METHOD PRIVATE M_MotionDynamicMove
VAR_INPUT
END_VAR
VAR_INST
	{attribute 'tc_no_symbol'}                	                			
	_fb_MovePosDynamic			: ARRAY [1..4] OF FB_ServoMotionDynamics;
	{attribute 'tc_no_symbol'}                	                			
	_enableDynamicMove			: BOOL;
	{attribute 'tc_no_symbol'}                	                			
	_Pos2MoveStart				: ST_MovePosition_SP;
	{attribute 'tc_no_symbol'}                	                			
	_CMD_MoveDynamicAbsStart	: ARRAY[1..4] OF MC_MOVEABSOLUTE;
	{attribute 'tc_no_symbol'}                	                			
	_CMD_MoveDynamicAbsEnd		: ARRAY[1..4] OF MC_MOVEABSOLUTE;
END_VAR
VAR_INST // added by the converter: edge detectors and wires of the graphical bodies
    _rt1, _rt2, _rt3, _rt4, _rt5, _rt6, _rt7, _rt8, _rt9, _rt10 : R_TRIG;
    _w1, _w2 : BOOL;
END_VAR
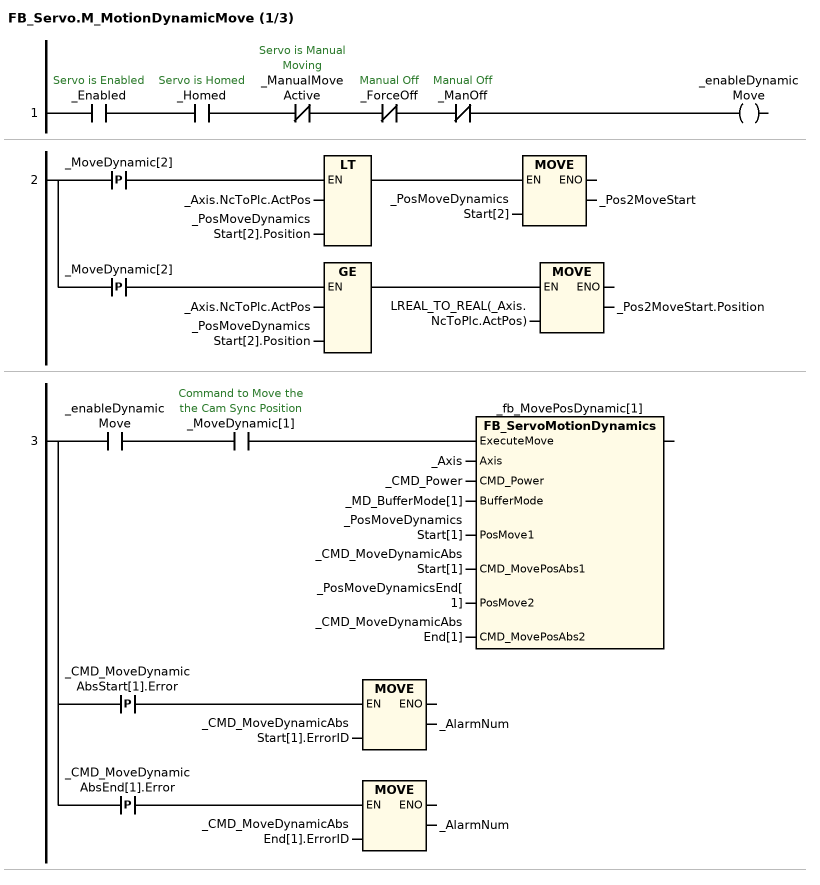
// NETWORK 1
//   _Enabled: Servo is Enabled
//   _Homed: Servo is Homed
//   _ManualMoveActive: Servo is Manual Moving
//   _ForceOff: Manual Off
//   _ManOff: Manual Off
_enableDynamicMove := _Enabled AND _Homed AND NOT _ManualMoveActive AND NOT _ForceOff AND NOT _ManOff;

// NETWORK 2
_rt1(CLK := _MoveDynamic[2]);
_w1 := _rt1.Q AND _Axis.NcToPlc.ActPos < _PosMoveDynamicsStart[2].Position;
IF _w1 THEN _Pos2MoveStart := _PosMoveDynamicsStart[2]; END_IF
_rt2(CLK := _MoveDynamic[2]);
_w2 := _rt2.Q AND _Axis.NcToPlc.ActPos >= _PosMoveDynamicsStart[2].Position;
IF _w2 THEN _Pos2MoveStart.Position := LREAL_TO_REAL(_Axis.NcToPlc.ActPos); END_IF

// NETWORK 3
//   _MoveDynamic[1]: Command to Move the the Cam Sync Position
_fb_MovePosDynamic[1](
    ExecuteMove := _enableDynamicMove AND _MoveDynamic[1],
    Axis := _Axis,
    CMD_Power := _CMD_Power,
    BufferMode := _MD_BufferMode[1],
    PosMove1 := _PosMoveDynamicsStart[1],
    CMD_MovePosAbs1 := _CMD_MoveDynamicAbsStart[1],
    PosMove2 := _PosMoveDynamicsEnd[1],
    CMD_MovePosAbs2 := _CMD_MoveDynamicAbsEnd[1]); // FB_ServoMotionDynamics
_rt3(CLK := _CMD_MoveDynamicAbsStart[1].Error);
IF _rt3.Q THEN _AlarmNum := _CMD_MoveDynamicAbsStart[1].ErrorID; END_IF
_rt4(CLK := _CMD_MoveDynamicAbsEnd[1].Error);
IF _rt4.Q THEN _AlarmNum := _CMD_MoveDynamicAbsEnd[1].ErrorID; END_IF

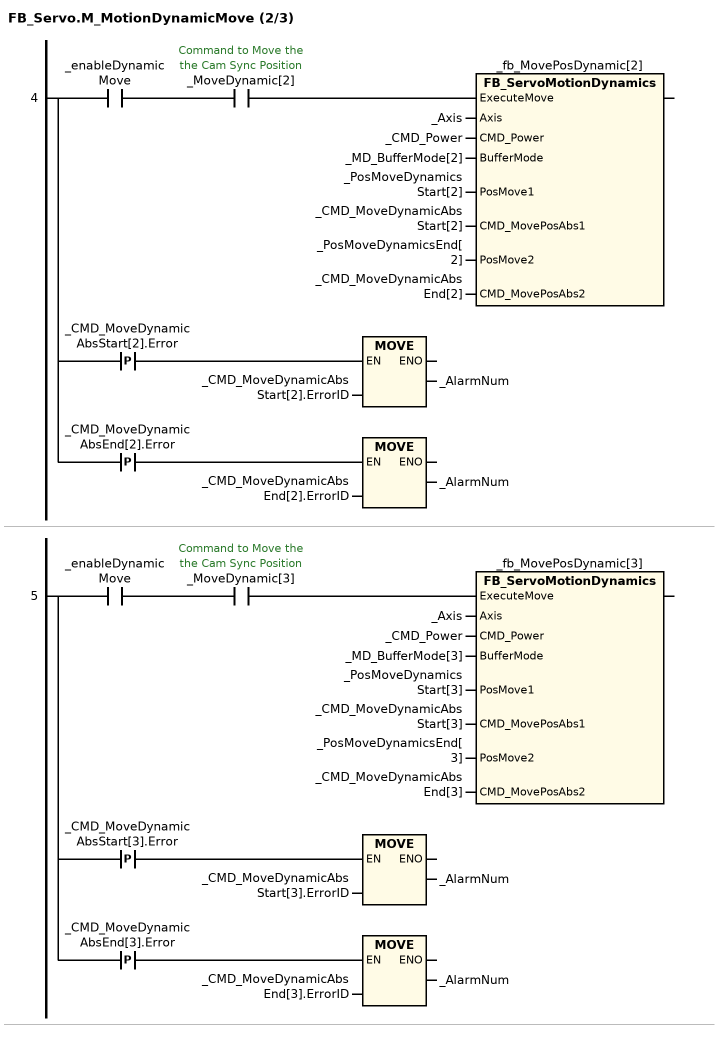
// NETWORK 4
//   _MoveDynamic[2]: Command to Move the the Cam Sync Position
_fb_MovePosDynamic[2](
    ExecuteMove := _enableDynamicMove AND _MoveDynamic[2],
    Axis := _Axis,
    CMD_Power := _CMD_Power,
    BufferMode := _MD_BufferMode[2],
    PosMove1 := _PosMoveDynamicsStart[2],
    CMD_MovePosAbs1 := _CMD_MoveDynamicAbsStart[2],
    PosMove2 := _PosMoveDynamicsEnd[2],
    CMD_MovePosAbs2 := _CMD_MoveDynamicAbsEnd[2]); // FB_ServoMotionDynamics
_rt5(CLK := _CMD_MoveDynamicAbsStart[2].Error);
IF _rt5.Q THEN _AlarmNum := _CMD_MoveDynamicAbsStart[2].ErrorID; END_IF
_rt6(CLK := _CMD_MoveDynamicAbsEnd[2].Error);
IF _rt6.Q THEN _AlarmNum := _CMD_MoveDynamicAbsEnd[2].ErrorID; END_IF

// NETWORK 5
//   _MoveDynamic[3]: Command to Move the the Cam Sync Position
_fb_MovePosDynamic[3](
    ExecuteMove := _enableDynamicMove AND _MoveDynamic[3],
    Axis := _Axis,
    CMD_Power := _CMD_Power,
    BufferMode := _MD_BufferMode[3],
    PosMove1 := _PosMoveDynamicsStart[3],
    CMD_MovePosAbs1 := _CMD_MoveDynamicAbsStart[3],
    PosMove2 := _PosMoveDynamicsEnd[3],
    CMD_MovePosAbs2 := _CMD_MoveDynamicAbsEnd[3]); // FB_ServoMotionDynamics
_rt7(CLK := _CMD_MoveDynamicAbsStart[3].Error);
IF _rt7.Q THEN _AlarmNum := _CMD_MoveDynamicAbsStart[3].ErrorID; END_IF
_rt8(CLK := _CMD_MoveDynamicAbsEnd[3].Error);
IF _rt8.Q THEN _AlarmNum := _CMD_MoveDynamicAbsEnd[3].ErrorID; END_IF

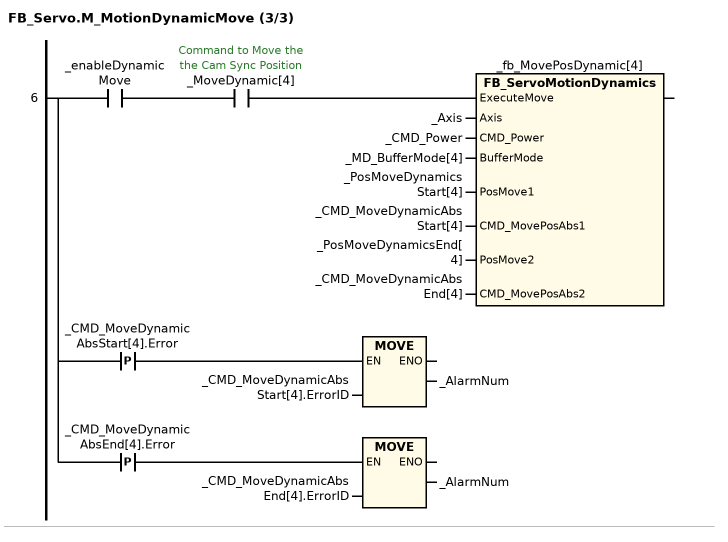
// NETWORK 6
//   _MoveDynamic[4]: Command to Move the the Cam Sync Position
_fb_MovePosDynamic[4](
    ExecuteMove := _enableDynamicMove AND _MoveDynamic[4],
    Axis := _Axis,
    CMD_Power := _CMD_Power,
    BufferMode := _MD_BufferMode[4],
    PosMove1 := _PosMoveDynamicsStart[4],
    CMD_MovePosAbs1 := _CMD_MoveDynamicAbsStart[4],
    PosMove2 := _PosMoveDynamicsEnd[4],
    CMD_MovePosAbs2 := _CMD_MoveDynamicAbsEnd[4]); // FB_ServoMotionDynamics
_rt9(CLK := _CMD_MoveDynamicAbsStart[4].Error);
IF _rt9.Q THEN _AlarmNum := _CMD_MoveDynamicAbsStart[4].ErrorID; END_IF
_rt10(CLK := _CMD_MoveDynamicAbsEnd[4].Error);
IF _rt10.Q THEN _AlarmNum := _CMD_MoveDynamicAbsEnd[4].ErrorID; END_IF
END_METHOD

METHOD PRIVATE M_MoveSuperImposed
VAR_INPUT
END_VAR
VAR_INST
	{attribute 'tc_no_symbol'}                	                			
	_enableSuperImposed					: BOOL;
	{attribute 'tc_no_symbol'}                	                			
	_CMD_MoveSuperImposed				: MC_MOVESUPERIMPOSED;
END_VAR
VAR_INST // added by the converter: edge detectors and wires of the graphical bodies
    _rt1 : R_TRIG;
END_VAR
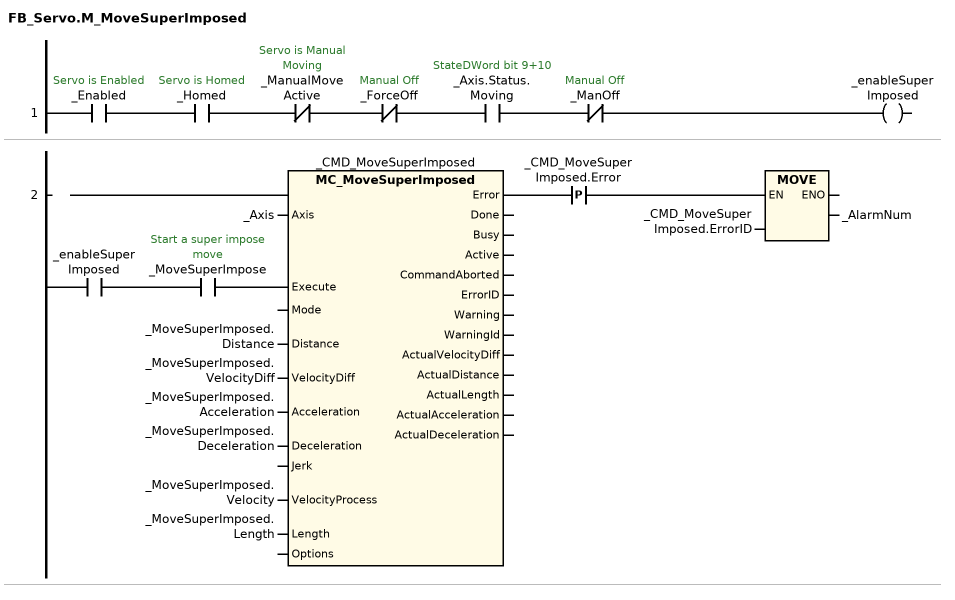
// NETWORK 1
//   _Enabled: Servo is Enabled
//   _Homed: Servo is Homed
//   _ManualMoveActive: Servo is Manual Moving
//   _ForceOff: Manual Off
//   _Axis.Status.Moving: StateDWord bit 9+10
//   _ManOff: Manual Off
_enableSuperImposed := _Enabled AND _Homed AND NOT _ManualMoveActive AND NOT _ForceOff AND _Axis.Status.Moving AND NOT _ManOff;

// NETWORK 2
//   _MoveSuperImpose: Start a super impose move
//   _MoveSuperImposed.Distance: Relative distance to catch up or fall back with the super imposed move
//   _MoveSuperImposed.VelocityDiff: Velocity Value of the catch up or fall back distance
//   _MoveSuperImposed.Acceleration: Accleration Value of Move
//   _MoveSuperImposed.Deceleration: Deceleration Value of Move
//   _MoveSuperImposed.Velocity: Velocity Value of Move without move super imposed
//   _MoveSuperImposed.Length: Length of the total move distance
_CMD_MoveSuperImposed(
    Axis := _Axis,
    Execute := _enableSuperImposed AND _MoveSuperImpose,
    Distance := _MoveSuperImposed.Distance,
    VelocityDiff := _MoveSuperImposed.VelocityDiff,
    Acceleration := _MoveSuperImposed.Acceleration,
    Deceleration := _MoveSuperImposed.Deceleration,
    VelocityProcess := _MoveSuperImposed.Velocity,
    Length := _MoveSuperImposed.Length); // MC_MoveSuperImposed
_rt1(CLK := _CMD_MoveSuperImposed.Error);
IF _CMD_MoveSuperImposed.Error AND _rt1.Q THEN _AlarmNum := _CMD_MoveSuperImposed.ErrorID; END_IF
END_METHOD

METHOD PRIVATE M_MoveToPosition
VAR_INPUT
END_VAR
VAR_INST
	{attribute 'tc_no_symbol'}                	                			
	_fb_MovePos							: ARRAY [1..4] OF FB_ServoMove;
	{attribute 'tc_no_symbol'}                	                			
	_fb_MovePosSync						: FB_ServoMove;
	{attribute 'tc_no_symbol'}                	                			
	_enableMove							: BOOL;
	{attribute 'tc_no_symbol'}                	                			
	_enableMoveHalt						: BOOL;
	{attribute 'tc_no_symbol'}                	                			
	_decelRateMoveHalt					: LREAL;
	{attribute 'tc_no_symbol'}                	                			
	_CMD_MovePosSyncAbs					: MC_MOVEABSOLUTE;
	{attribute 'tc_no_symbol'}                	                			
	_CMD_MovePosSyncMod					: MC_MOVEMODULO;
	{attribute 'tc_no_symbol'}                	                			
	_CMD_MovePosSyncRel					: MC_MOVERELATIVE;
	{attribute 'tc_no_symbol'}                	                			
	_CMD_MoveHalt						: MC_HALT;
	{attribute 'tc_no_symbol'}                	                			
	_CMD_MovePosAbs						: ARRAY[1..4] OF MC_MOVEABSOLUTE;
	{attribute 'tc_no_symbol'}                	                			
	_CMD_MovePosMod						: ARRAY[1..4] OF MC_MOVEMODULO;
	{attribute 'tc_no_symbol'}                	                			
	_CMD_MovePosRel						: ARRAY[1..4] OF MC_MOVERELATIVE;
	{attribute 'tc_no_symbol'}                	                			
	_R_Trig								: ARRAY[0..3] OF R_TRIG;
END_VAR
VAR_INST // added by the converter: edge detectors and wires of the graphical bodies
    _rt1, _rt2, _rt3, _rt4, _rt5, _rt6, _rt7, _rt8, _rt9, _rt10, _rt11, _rt12, _rt13, _rt14, _rt15, _rt16 : R_TRIG;
END_VAR
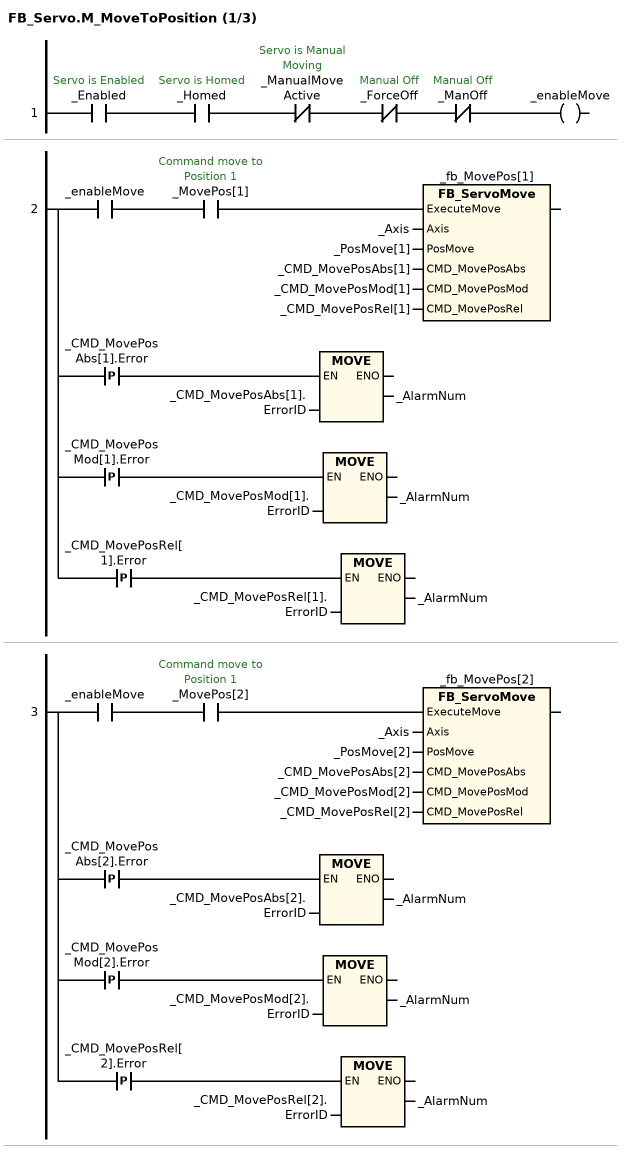
// NETWORK 1
//   _Enabled: Servo is Enabled
//   _Homed: Servo is Homed
//   _ManualMoveActive: Servo is Manual Moving
//   _ForceOff: Manual Off
//   _ManOff: Manual Off
_enableMove := _Enabled AND _Homed AND NOT _ManualMoveActive AND NOT _ForceOff AND NOT _ManOff;

// NETWORK 2
//   _MovePos[1]: Command move to Position 1
//   _PosMove[1]: Position 1 Move Setpoints
_fb_MovePos[1](
    ExecuteMove := _enableMove AND _MovePos[1],
    Axis := _Axis,
    PosMove := _PosMove[1],
    CMD_MovePosAbs := _CMD_MovePosAbs[1],
    CMD_MovePosMod := _CMD_MovePosMod[1],
    CMD_MovePosRel := _CMD_MovePosRel[1]); // FB_ServoMove
_rt1(CLK := _CMD_MovePosAbs[1].Error);
IF _rt1.Q THEN _AlarmNum := _CMD_MovePosAbs[1].ErrorID; END_IF
_rt2(CLK := _CMD_MovePosMod[1].Error);
IF _rt2.Q THEN _AlarmNum := _CMD_MovePosMod[1].ErrorID; END_IF
_rt3(CLK := _CMD_MovePosRel[1].Error);
IF _rt3.Q THEN _AlarmNum := _CMD_MovePosRel[1].ErrorID; END_IF

// NETWORK 3
//   _MovePos[2]: Command move to Position 1
//   _PosMove[2]: Position 1 Move Setpoints
_fb_MovePos[2](
    ExecuteMove := _enableMove AND _MovePos[2],
    Axis := _Axis,
    PosMove := _PosMove[2],
    CMD_MovePosAbs := _CMD_MovePosAbs[2],
    CMD_MovePosMod := _CMD_MovePosMod[2],
    CMD_MovePosRel := _CMD_MovePosRel[2]); // FB_ServoMove
_rt4(CLK := _CMD_MovePosAbs[2].Error);
IF _rt4.Q THEN _AlarmNum := _CMD_MovePosAbs[2].ErrorID; END_IF
_rt5(CLK := _CMD_MovePosMod[2].Error);
IF _rt5.Q THEN _AlarmNum := _CMD_MovePosMod[2].ErrorID; END_IF
_rt6(CLK := _CMD_MovePosRel[2].Error);
IF _rt6.Q THEN _AlarmNum := _CMD_MovePosRel[2].ErrorID; END_IF

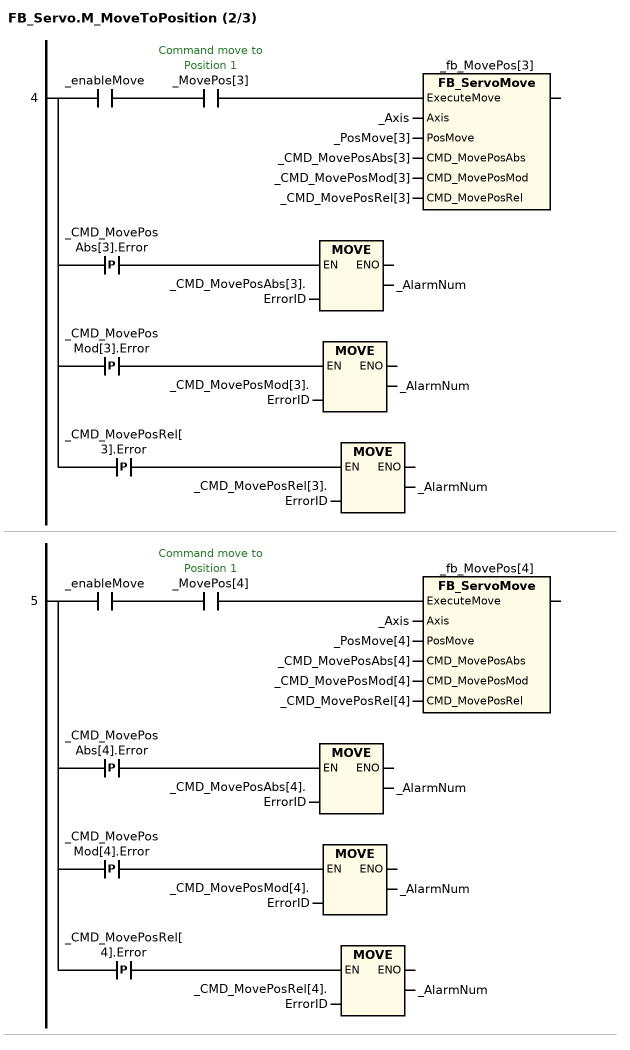
// NETWORK 4
//   _MovePos[3]: Command move to Position 1
//   _PosMove[3]: Position 1 Move Setpoints
_fb_MovePos[3](
    ExecuteMove := _enableMove AND _MovePos[3],
    Axis := _Axis,
    PosMove := _PosMove[3],
    CMD_MovePosAbs := _CMD_MovePosAbs[3],
    CMD_MovePosMod := _CMD_MovePosMod[3],
    CMD_MovePosRel := _CMD_MovePosRel[3]); // FB_ServoMove
_rt7(CLK := _CMD_MovePosAbs[3].Error);
IF _rt7.Q THEN _AlarmNum := _CMD_MovePosAbs[3].ErrorID; END_IF
_rt8(CLK := _CMD_MovePosMod[3].Error);
IF _rt8.Q THEN _AlarmNum := _CMD_MovePosMod[3].ErrorID; END_IF
_rt9(CLK := _CMD_MovePosRel[3].Error);
IF _rt9.Q THEN _AlarmNum := _CMD_MovePosRel[3].ErrorID; END_IF

// NETWORK 5
//   _MovePos[4]: Command move to Position 1
//   _PosMove[4]: Position 1 Move Setpoints
_fb_MovePos[4](
    ExecuteMove := _enableMove AND _MovePos[4],
    Axis := _Axis,
    PosMove := _PosMove[4],
    CMD_MovePosAbs := _CMD_MovePosAbs[4],
    CMD_MovePosMod := _CMD_MovePosMod[4],
    CMD_MovePosRel := _CMD_MovePosRel[4]); // FB_ServoMove
_rt10(CLK := _CMD_MovePosAbs[4].Error);
IF _rt10.Q THEN _AlarmNum := _CMD_MovePosAbs[4].ErrorID; END_IF
_rt11(CLK := _CMD_MovePosMod[4].Error);
IF _rt11.Q THEN _AlarmNum := _CMD_MovePosMod[4].ErrorID; END_IF
_rt12(CLK := _CMD_MovePosRel[4].Error);
IF _rt12.Q THEN _AlarmNum := _CMD_MovePosRel[4].ErrorID; END_IF

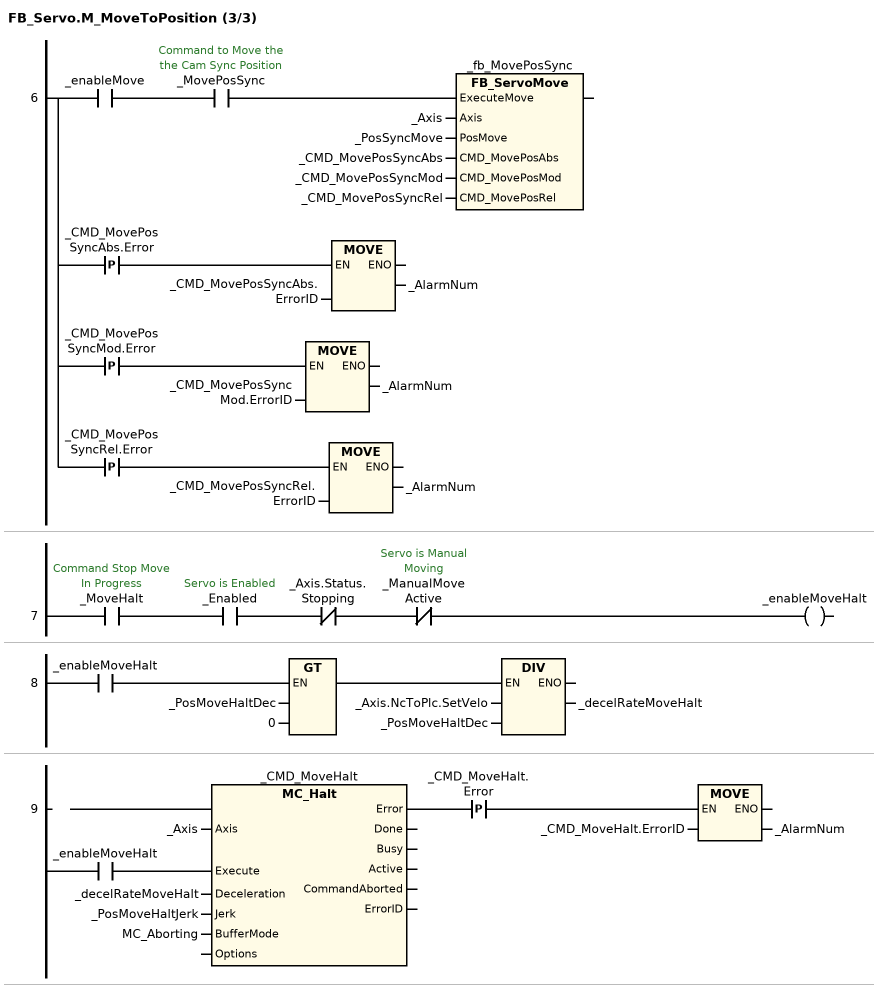
// NETWORK 6
//   _MovePosSync: Command to Move the the Cam Sync Position
//   _PosSyncMove: Sync Position Move Setpoints
_fb_MovePosSync(
    ExecuteMove := _enableMove AND _MovePosSync,
    Axis := _Axis,
    PosMove := _PosSyncMove,
    CMD_MovePosAbs := _CMD_MovePosSyncAbs,
    CMD_MovePosMod := _CMD_MovePosSyncMod,
    CMD_MovePosRel := _CMD_MovePosSyncRel); // FB_ServoMove
_rt13(CLK := _CMD_MovePosSyncAbs.Error);
IF _rt13.Q THEN _AlarmNum := _CMD_MovePosSyncAbs.ErrorID; END_IF
_rt14(CLK := _CMD_MovePosSyncMod.Error);
IF _rt14.Q THEN _AlarmNum := _CMD_MovePosSyncMod.ErrorID; END_IF
_rt15(CLK := _CMD_MovePosSyncRel.Error);
IF _rt15.Q THEN _AlarmNum := _CMD_MovePosSyncRel.ErrorID; END_IF

// NETWORK 7
//   _MoveHalt: Command Stop Move In Progress
//   _Enabled: Servo is Enabled
//   _ManualMoveActive: Servo is Manual Moving
_enableMoveHalt := _MoveHalt AND _Enabled AND NOT _Axis.Status.Stopping AND NOT _ManualMoveActive;

// NETWORK 8
//   _PosMoveHaltDec: Positional Move Halt Deceration
IF _enableMoveHalt AND _PosMoveHaltDec > 0 THEN
    _decelRateMoveHalt := _Axis.NcToPlc.SetVelo / _PosMoveHaltDec;
END_IF

// NETWORK 9
//   _PosMoveHaltJerk: Positional Move Halt Jerk
_CMD_MoveHalt(
    Axis := _Axis,
    Execute := _enableMoveHalt,
    Deceleration := _decelRateMoveHalt,
    Jerk := _PosMoveHaltJerk,
    BufferMode := MC_Aborting); // MC_Halt
_rt16(CLK := _CMD_MoveHalt.Error);
IF _CMD_MoveHalt.Error AND _rt16.Q THEN _AlarmNum := _CMD_MoveHalt.ErrorID; END_IF
END_METHOD

METHOD PRIVATE M_SettingsControl
VAR_INPUT
END_VAR
VAR_INST
	{attribute 'tc_no_symbol'}                	                			
	_homeOffsetPosition_Used			: LREAL;
	{attribute 'tc_no_symbol'}                	                			
	_maxPositionLag_Used				: LREAL;			
	{attribute 'tc_no_symbol'}                	                			
	_maxPositionLagTime_Used			: LREAL;	
	{attribute 'tc_no_symbol'}                	                					
	_softPositionLimitMaxActive_Used	: BOOL;				
	{attribute 'tc_no_symbol'}                	                			
	_softPositionLimitMinActive_Used	: BOOL;		
	{attribute 'tc_no_symbol'}                	                					
	_softPositionLimitMax_Used			: LREAL;	
	{attribute 'tc_no_symbol'}                	                					
	_softPositionLimitMin_Used			: LREAL;
	{attribute 'tc_no_symbol'}                	
	_MaxDriveOffDelay_Used				: DINT;
	{attribute 'tc_no_symbol'}   
	_HomeMode_Used						: INT;   
	_HomingCamSearchDirection_Used		: BOOL;  
	_HomingSyncSearchDirection_Used		: BOOL;               			
	_MaxDeceleration					: LREAL;
	{attribute 'tc_no_symbol'}                	                			
	_r_SetWrite_Trig					: ARRAY[0..10] OF R_TRIG;
	{attribute 'tc_no_symbol'}                	                			
	_r_SetRead_Trig						: ARRAY[0..10] OF R_TRIG;
	{attribute 'tc_no_symbol'}                	                			
	_r_Get_Trig							: R_TRIG;
	{attribute 'tc_no_symbol'}                	                			
	_CMD_ReadMaxDecelADS				: ADSREAD;
	{attribute 'tc_no_symbol'}                	                			
	_CMD_WriteParameterSet				: ARRAY[0..10] OF MC_WRITEPARAMETER;
	{attribute 'tc_no_symbol'}                	                			
	_CMD_ReadParameterSet				: ARRAY[0..10] OF MC_READPARAMETER;
	{attribute 'tc_no_symbol'}                	                			
	_CMD_ReadParameterGet				: ARRAY[0..10] OF MC_READPARAMETER;   
	{attribute 'tc_no_symbol'}   			
	_i									: USINT;
	{attribute 'tc_no_symbol'}                	                			
	_r_trig								: ARRAY[0..3] OF R_TRIG;
END_VAR
// Parameter Set
IF _Axis.Status.Disabled AND NOT Control.SystemTime.FirstCycle THEN
	
	//Set Torque Limits
	IF (_ManHome.Enabled OR _AutoHome) THEN
		_ServoTorqueLimit := F_CheckIndexBounds_UINT(10,100,_HomingTorqueLimit)*10;
	ELSE
		_ServoTorqueLimit := F_CheckIndexBounds_UINT(10,100,_NormalTorqueLimit)*10;
	END_IF;

	// Home Position Offset Value Set
	IF _Settings.HomeOffsetPosition <> _homeOffsetPosition_Used THEN
		_homeOffsetPosition_Used := _Settings.HomeOffsetPosition;
	END_IF
	
	// Maximum Position Lag Value Set
	_r_SetWrite_Trig[0](CLK:= _Settings.MaxPositionLag <> _maxPositionLag_Used);
	_CMD_WriteParameterSet[0](Axis := _Axis, Execute := _r_SetWrite_Trig[0].Q, ParameterNumber := MC_AxisParameter.MaxPositionLag,Value := _Settings.MaxPositionLag);
	_r_SetRead_Trig[0](CLK:= _CMD_WriteParameterSet[0].Done);
	_CMD_ReadParameterSet[0](Axis := _Axis, Enable := _r_SetRead_Trig[0].Q, ParameterNumber := MC_AxisParameter.MaxPositionLag,ReadMode := E_ReadMode.READMODE_ONCE);
	IF _CMD_ReadParameterSet[0].Valid THEN 
		_maxPositionLag_Used := _CMD_ReadParameterSet[0].Value; 
	END_IF

	// Maximum Position Lag Filter Time Set
	_r_SetWrite_Trig[1](CLK:=_Settings.MaxPositionLagTime <> _maxPositionLagTime_Used);
	_CMD_WriteParameterSet[1](Axis := _Axis, Execute := _r_SetWrite_Trig[1].Q, ParameterNumber := MC_AxisParameter.AxisMaxPosLagFilterTime, Value := _Settings.MaxPositionLagTime);
	_r_SetRead_Trig[1](CLK:= _CMD_WriteParameterSet[1].Done);
	_CMD_ReadParameterSet[1](Axis := _Axis, Enable := _r_SetRead_Trig[1].Q, ParameterNumber := MC_AxisParameter.AxisMaxPosLagFilterTime, ReadMode := E_ReadMode.READMODE_ONCE);
	IF _CMD_ReadParameterSet[1].Valid THEN 
		_maxPositionLagTime_Used := _CMD_ReadParameterSet[1].Value; 
	END_IF

	// Soft Position Limit Maximum Active Set
	_r_SetWrite_Trig[2](CLK:=_Settings.SoftPositionLimitMaxActive <> _softPositionLimitMaxActive_Used);
	_CMD_WriteParameterSet[2](Axis := _Axis, Execute := _r_SetWrite_Trig[2].Q, ParameterNumber := MC_AxisParameter.AxisEnMaxSoftPosLimit,Value := BOOL_TO_LREAL(_Settings.SoftPositionLimitMaxActive));
	_r_SetRead_Trig[2](CLK:= _CMD_WriteParameterSet[2].Done);
	_CMD_ReadParameterSet[2](Axis := _Axis, Enable := _r_SetRead_Trig[2].Q, ParameterNumber := MC_AxisParameter.AxisEnMaxSoftPosLimit, ReadMode := E_ReadMode.READMODE_ONCE);
	IF _CMD_ReadParameterSet[2].Valid THEN 
		_softPositionLimitMaxActive_Used := LREAL_TO_BOOL(_CMD_ReadParameterSet[2].Value); 
	END_IF
	
	// Soft Position Limit Minimum Active Set
	_r_SetWrite_Trig[3](CLK:=_Settings.SoftPositionLimitMinActive <> _softPositionLimitMinActive_Used);
	_CMD_WriteParameterSet[3](Axis := _Axis, Execute := _r_SetWrite_Trig[3].Q, ParameterNumber := MC_AxisParameter.AxisEnMinSoftPosLimit, Value := BOOL_TO_LREAL(_Settings.SoftPositionLimitMinActive));
	_r_SetRead_Trig[3](CLK:= _CMD_WriteParameterSet[3].Done);
	_CMD_ReadParameterSet[3](Axis := _Axis, Enable := _r_SetRead_Trig[3].Q, ParameterNumber := MC_AxisParameter.AxisEnMinSoftPosLimit, ReadMode := E_ReadMode.READMODE_ONCE);
	IF _CMD_ReadParameterSet[3].Valid THEN 
		_softPositionLimitMinActive_Used := LREAL_TO_BOOL(_CMD_ReadParameterSet[3].Value); 
	END_IF
	
	// Soft Position Limit Maximum Value Set
	_r_SetWrite_Trig[4](CLK:=_Settings.SoftPositionLimitMax <> _softPositionLimitMax_Used);
	_CMD_WriteParameterSet[4](Axis := _Axis, Execute := _r_SetWrite_Trig[4].Q, ParameterNumber := MC_AxisParameter.AxisMaxSoftPosLimit, Value := _Settings.SoftPositionLimitMax);
	_r_SetRead_Trig[4](CLK:=_CMD_WriteParameterSet[4].Done);
	_CMD_ReadParameterSet[4](Axis := _Axis, Enable := _r_SetRead_Trig[4].Q, ParameterNumber := MC_AxisParameter.AxisMaxSoftPosLimit, ReadMode := E_ReadMode.READMODE_ONCE);
	IF _CMD_ReadParameterSet[4].Valid THEN 
		_softPositionLimitMax_Used := _CMD_ReadParameterSet[4].Value; 
	END_IF
	
	// Soft Position Limit Minimum Value Set
	_r_SetWrite_Trig[5](CLK:=_Settings.SoftPositionLimitMin <> _softPositionLimitMin_Used);
	_CMD_WriteParameterSet[5](Axis := _Axis, Execute := _r_SetWrite_Trig[5].Q, ParameterNumber := MC_AxisParameter.AxisMinSoftPosLimit, Value := _Settings.SoftPositionLimitMin);
	_r_SetRead_Trig[5](CLK:=_CMD_WriteParameterSet[5].Done);
	_CMD_ReadParameterSet[5](Axis := _Axis, Enable := _r_SetRead_Trig[5].Q, ParameterNumber := MC_AxisParameter.AxisMinSoftPosLimit, ReadMode := E_ReadMode.READMODE_ONCE);
	IF _CMD_ReadParameterSet[5].Valid THEN 
		_softPositionLimitMin_Used := _CMD_ReadParameterSet[5].Value; 
	END_IF
	
	// Homing mode direction set - FALSE = FWD	
	CASE _HomeMode OF
		0: _Settings.HomingCamSearchDirection := TRUE; _Settings.HomingSyncSearchDirection := FALSE;
		1: _Settings.HomingCamSearchDirection := FALSE; _Settings.HomingSyncSearchDirection := FALSE;
		2: _Settings.HomingCamSearchDirection := FALSE; _Settings.HomingSyncSearchDirection := TRUE;
	END_CASE
	
	_r_SetWrite_Trig[6](CLK:=_Settings.HomingCamSearchDirection <> _HomingCamSearchDirection_Used);
	_CMD_WriteParameterSet[6](Axis := _Axis, Execute := _r_SetWrite_Trig[6].Q, ParameterNumber := MC_AxisParameter.AxisEncoderHomingInvDirCamSearch, Value := BOOL_TO_LREAL(_Settings.HomingCamSearchDirection));
	_r_SetRead_Trig[6](CLK:=_CMD_WriteParameterSet[6].Done);
	_CMD_ReadParameterSet[6](Axis := _Axis, Enable := _r_SetRead_Trig[6].Q, ParameterNumber := MC_AxisParameter.AxisEncoderHomingInvDirCamSearch, ReadMode := E_ReadMode.READMODE_ONCE);
	IF _CMD_ReadParameterSet[6].Valid THEN 
		_HomingCamSearchDirection_Used		:= LREAL_TO_BOOL(_CMD_ReadParameterSet[6].Value); 
	END_IF;
	
	_r_SetWrite_Trig[7](CLK:=_Settings.HomingSyncSearchDirection <> _HomingSyncSearchDirection_Used);
	_CMD_WriteParameterSet[7](Axis := _Axis, Execute := _r_SetWrite_Trig[6].Q, ParameterNumber := MC_AxisParameter.AxisEncoderHomingInvDirSyncSearch, Value := BOOL_TO_LREAL(_Settings.HomingSyncSearchDirection));
	_r_SetRead_Trig[7](CLK:=_CMD_WriteParameterSet[7].Done);
	_CMD_ReadParameterSet[7](Axis := _Axis, Enable := _r_SetRead_Trig[6].Q, ParameterNumber := MC_AxisParameter.AxisEncoderHomingInvDirSyncSearch, ReadMode := E_ReadMode.READMODE_ONCE);
	IF _CMD_ReadParameterSet[7].Valid THEN
		_HomingSyncSearchDirection_Used		:= LREAL_TO_BOOL(_CMD_ReadParameterSet[7].Value); 
	END_IF	
END_IF

// Parameter Get
_r_Get_Trig(CLK:= _UpdateDriveParameters OR Control.SystemTime.FirstCycle);

// Drive Status
_DriveStatus :=  F_ConvWordToSTAX5000DriveStatus(wDriveStatus:= _DriveStatusWord);

// Maximum Deceleration
_CMD_ReadMaxDecelADS(NETID := '',PORT := 501,IDXGRP := 16#00004002,IDXOFFS := 16#000000F2,LEN := 8,DESTADDR := ADR(_MaxDeceleration),READ := _r_Get_Trig.Q,TMOUT := ,BUSY => ,ERR => ,ERRID => ,);
_MaximumDeceleration := _MaxDeceleration;

// Maximum Position Lag Value Set
_CMD_ReadParameterGet[0](Axis := _Axis, Enable := _r_Get_Trig.Q, ParameterNumber := MC_AxisParameter.AxisMaxPosLagValue,ReadMode := E_ReadMode.READMODE_ONCE);
IF _CMD_ReadParameterGet[0].Valid THEN 
	_Settings.MaxPositionLag := _CMD_ReadParameterGet[0].Value; 
END_IF

// Maximum Position Lag Filter Time Get
_CMD_ReadParameterGet[1](Axis := _Axis, Enable := _r_Get_Trig.Q, ParameterNumber := MC_AxisParameter.AxisMaxPosLagFilterTime,ReadMode := E_ReadMode.READMODE_ONCE);
IF _CMD_ReadParameterGet[1].Valid THEN 
	_Settings.MaxPositionLagTime := _CMD_ReadParameterGet[1].Value; 
END_IF

// Soft Position Limit Maximum Active Get
_CMD_ReadParameterGet[2](Axis := _Axis, Enable := _r_Get_Trig.Q, ParameterNumber := MC_AxisParameter.AxisEnMaxSoftPosLimit,ReadMode := E_ReadMode.READMODE_ONCE);
IF _CMD_ReadParameterGet[2].Valid THEN 
	_Settings.SoftPositionLimitMaxActive := LREAL_TO_BOOL(_CMD_ReadParameterGet[2].Value); 
END_IF

// Soft Position Limit Minimum Active Get
_CMD_ReadParameterGet[3](Axis := _Axis, Enable := _r_Get_Trig.Q, ParameterNumber := MC_AxisParameter.AxisEnMinSoftPosLimit,ReadMode := E_ReadMode.READMODE_ONCE);
IF _CMD_ReadParameterGet[3].Valid THEN 
	_Settings.SoftPositionLimitMinActive := LREAL_TO_BOOL(_CMD_ReadParameterGet[3].Value); 
END_IF

// Soft Position Limit Maximum Value Get
_CMD_ReadParameterGet[4](Axis := _Axis, Enable := _r_Get_Trig.Q, ParameterNumber := MC_AxisParameter.AxisMaxSoftPosLimit,ReadMode := E_ReadMode.READMODE_ONCE);
IF _CMD_ReadParameterGet[4].Valid THEN 
	_Settings.SoftPositionLimitMax := _CMD_ReadParameterGet[4].Value; 
END_IF

// Soft Position Limit Minimum Value Get
_CMD_ReadParameterGet[5](Axis := _Axis, Enable := _r_Get_Trig.Q, ParameterNumber := MC_AxisParameter.AxisMinSoftPosLimit,ReadMode := E_ReadMode.READMODE_ONCE);
IF _CMD_ReadParameterGet[5].Valid THEN 
	_Settings.SoftPositionLimitMin := _CMD_ReadParameterGet[5].Value; 
END_IF

// Modulo Factor Value Get
_CMD_ReadParameterGet[6](Axis := _Axis, Enable := _r_Get_Trig.Q, ParameterNumber := MC_AxisParameter.AxisEncoderModuloValue,ReadMode := E_ReadMode.READMODE_ONCE);
IF _CMD_ReadParameterGet[6].Valid THEN 
	_Settings.ModuloFactor := _CMD_ReadParameterGet[6].Value; 
END_IF

//Check for Function Block Errors
_r_trig[0](CLK:=_CMD_ReadMaxDecelADS.ERR);	
IF _r_trig[0].Q THEN _AlarmNum := _CMD_ReadMaxDecelADS.ERRID; END_IF

FOR _i := 0 TO 10 BY 1 DO
 	_r_trig[1](CLK:=_CMD_WriteParameterSet[_i].Error);	
	IF _r_trig[1].Q THEN _AlarmNum := _CMD_WriteParameterSet[_i].ErrorID;END_IF
	_r_trig[2](CLK:=_CMD_ReadParameterSet[_i].Error);	
	IF _r_trig[2].Q THEN _AlarmNum := _CMD_ReadParameterSet[_i].ErrorID;END_IF
    _r_trig[3](CLK:=_CMD_ReadParameterGet[_i].Error);
	IF _r_trig[3].Q THEN _AlarmNum := _CMD_ReadParameterGet[_i].ErrorID;END_IF
END_FOR
END_METHOD

METHOD PRIVATE M_StateControl
VAR_INPUT
END_VAR
VAR_INST
	{attribute 'tc_no_symbol'}                	                			
	_StepTimerET						: REAL;
	{attribute 'tc_no_symbol'}                	                			
	_StepTimerPT						: ARRAY[0..20] OF REAL;
	{attribute 'tc_no_symbol'}                	                			
	_StepTimerDN						: BOOL;
	{attribute 'tc_no_symbol'}                	                			
	_last_Step							: DINT;					

END_VAR
VAR_INST // added by the converter: edge detectors and wires of the graphical bodies
    _w1 : BOOL;
END_VAR
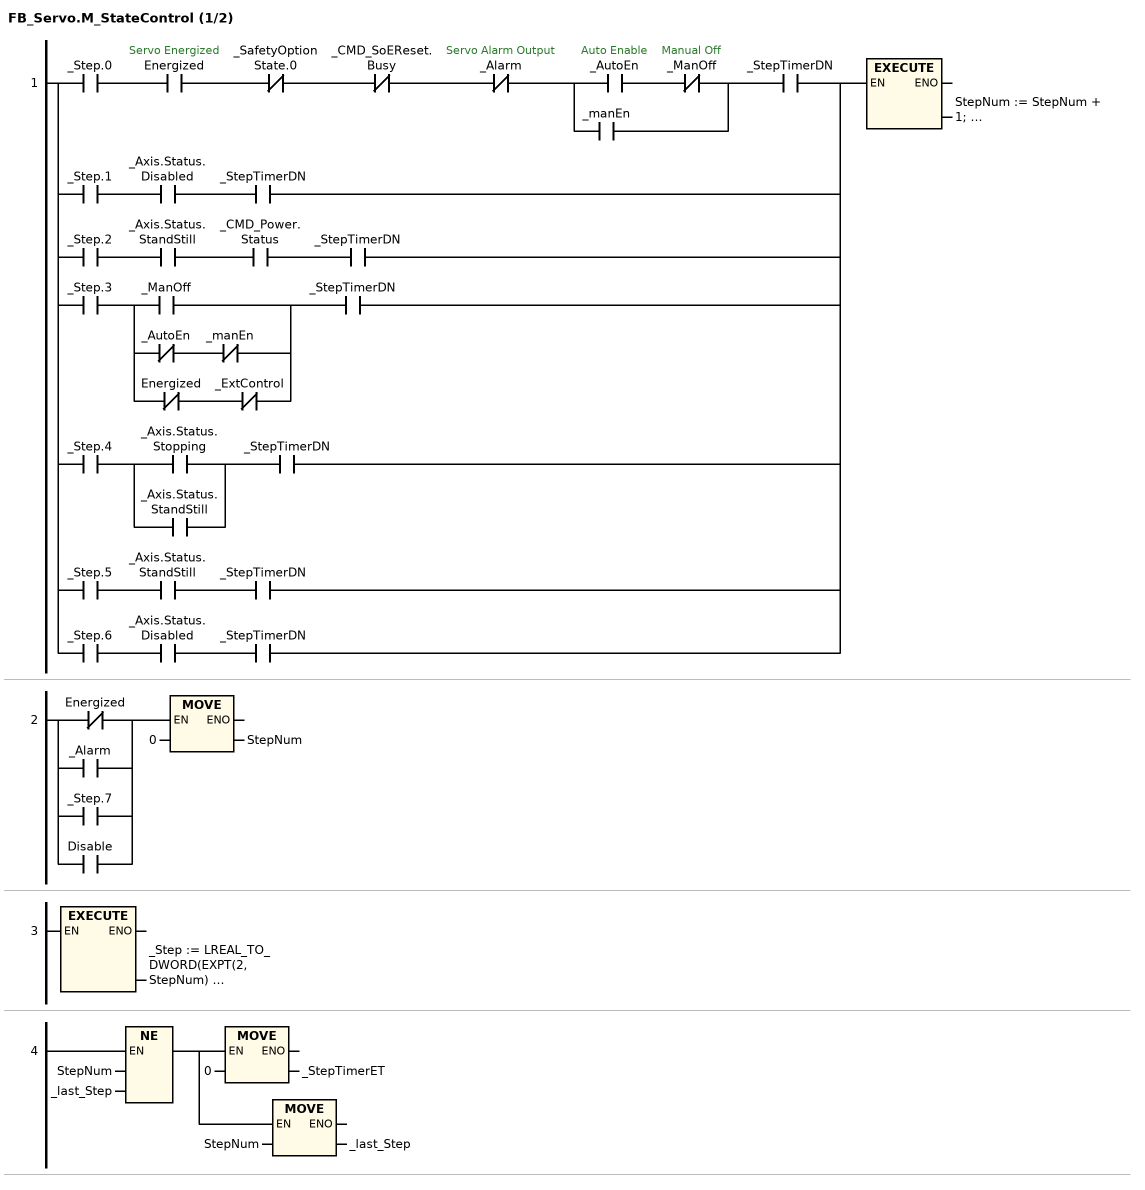
// NETWORK 1
//   Energized: Servo Energized
//   _Alarm: Servo Alarm Output
//   _AutoEn: Auto Enable
//   _ManOff: Manual Off
IF _Step.0 AND Energized AND NOT _SafetyOptionState.0 AND NOT _CMD_SoEReset.Busy AND NOT _Alarm AND (_AutoEn AND NOT _ManOff OR _manEn) AND _StepTimerDN OR _Step.1 AND _Axis.Status.Disabled AND _StepTimerDN OR _Step.2 AND _Axis.Status.StandStill AND _CMD_Power.Status AND _StepTimerDN OR _Step.3 AND (_ManOff OR NOT _AutoEn AND NOT _manEn OR NOT Energized AND NOT _ExtControl) AND _StepTimerDN OR _Step.4 AND (_Axis.Status.Stopping OR _Axis.Status.StandStill) AND _StepTimerDN OR _Step.5 AND _Axis.Status.StandStill AND _StepTimerDN OR _Step.6 AND _Axis.Status.Disabled AND _StepTimerDN THEN
    StepNum := StepNum + 1;
END_IF

// NETWORK 2
//   StepNum: Servo State Control Step Number Output
IF NOT Energized OR _Alarm OR _Step.7 OR Disable THEN StepNum := 0; END_IF

// NETWORK 3
_Step := LREAL_TO_DWORD(EXPT(2, StepNum));

// NETWORK 4
//   StepNum: Servo State Control Step Number Output
_w1 := StepNum <> _last_Step;
IF _w1 THEN _StepTimerET := 0; END_IF
IF _w1 THEN _last_Step := StepNum; END_IF

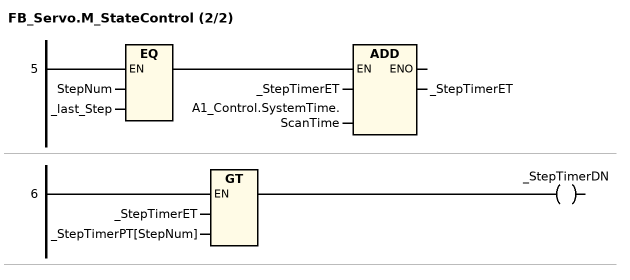
// NETWORK 5
//   StepNum: Servo State Control Step Number Output
//   A1_Control.SystemTime.ScanTime: Last scan time (Seconds)
IF StepNum = _last_Step THEN _StepTimerET := _StepTimerET + A1_Control.SystemTime.ScanTime; END_IF

// NETWORK 6
_StepTimerDN := _StepTimerET > _StepTimerPT[StepNum];
END_METHOD

METHOD PRIVATE M_StateOutputs
VAR_INPUT
END_VAR
VAR_INST
	{attribute 'tc_no_symbol'}                	                			
	_power				: BOOL;
	{attribute 'tc_no_symbol'}                	                			
	_decelRate			: LREAL;
	{attribute 'tc_no_symbol'}                	                			
	_CMD_Reset			: MC_RESET;
	{attribute 'tc_no_symbol'}                	                			
	_CMD_Stop			: MC_STOP;
END_VAR
VAR_INST // added by the converter: edge detectors and wires of the graphical bodies
    _rt1, _rt2, _rt3, _rt4 : R_TRIG;
    _w1 : BOOL;
END_VAR
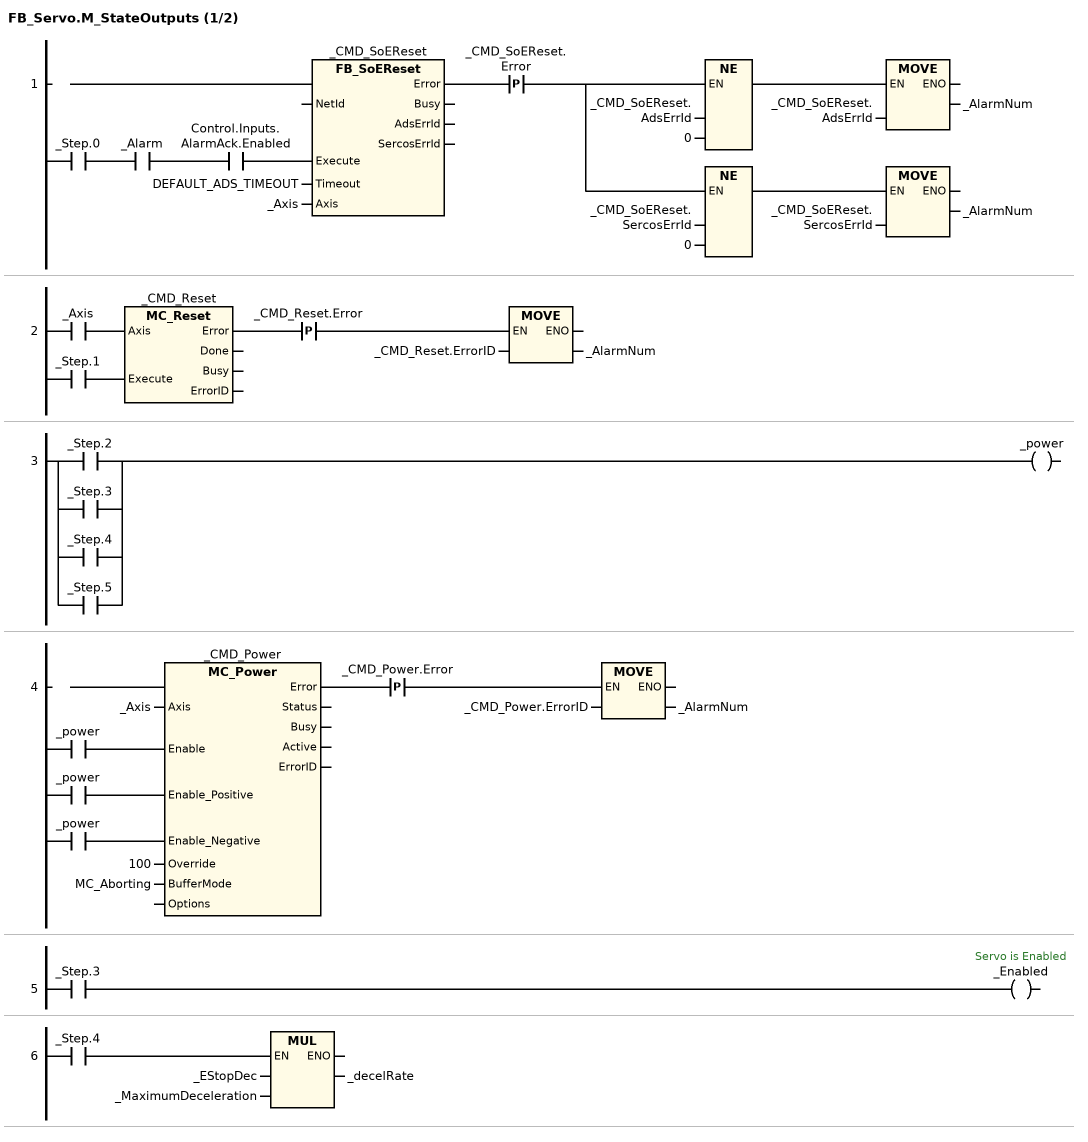
// NETWORK 1
_CMD_SoEReset(
    Execute := _Step.0 AND _Alarm AND Control.Inputs.AlarmAck.Enabled,
    Timeout := DEFAULT_ADS_TIMEOUT,
    Axis := _Axis); // FB_SoEReset
_rt1(CLK := _CMD_SoEReset.Error);
_w1 := _CMD_SoEReset.Error AND _rt1.Q;
IF _w1 AND _CMD_SoEReset.AdsErrId <> 0 THEN _AlarmNum := _CMD_SoEReset.AdsErrId; END_IF
IF _w1 AND _CMD_SoEReset.SercosErrId <> 0 THEN _AlarmNum := _CMD_SoEReset.SercosErrId; END_IF

// NETWORK 2
_CMD_Reset(Axis := _Axis, Execute := _Step.1); // MC_Reset
_rt2(CLK := _CMD_Reset.Error);
IF _CMD_Reset.Error AND _rt2.Q THEN _AlarmNum := _CMD_Reset.ErrorID; END_IF

// NETWORK 3
_power := _Step.2 OR _Step.3 OR _Step.4 OR _Step.5;

// NETWORK 4
_CMD_Power(
    Axis := _Axis,
    Enable := _power,
    Enable_Positive := _power,
    Enable_Negative := _power,
    Override := 100,
    BufferMode := MC_Aborting); // MC_Power
_rt3(CLK := _CMD_Power.Error);
IF _CMD_Power.Error AND _rt3.Q THEN _AlarmNum := _CMD_Power.ErrorID; END_IF

// NETWORK 5
//   _Enabled: Servo is Enabled
_Enabled := _Step.3;

// NETWORK 6
//   _EStopDec: EStop Deceleration Percentage
//   _MaximumDeceleration: Maximum Deceleration of the System
IF _Step.4 THEN _decelRate := _EStopDec * _MaximumDeceleration; END_IF

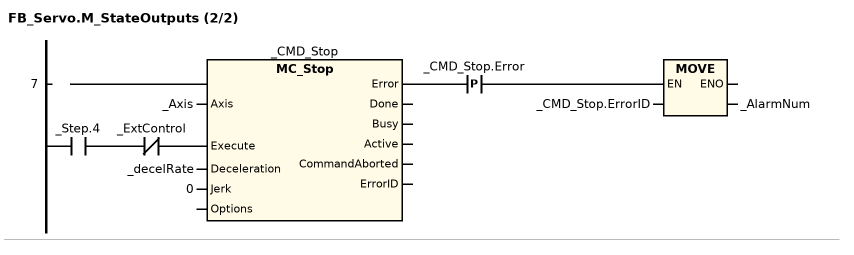
// NETWORK 7
_CMD_Stop(Axis := _Axis, Execute := _Step.4 AND NOT _ExtControl, Deceleration := _decelRate, Jerk := 0); // MC_Stop
_rt4(CLK := _CMD_Stop.Error);
IF _CMD_Stop.Error AND _rt4.Q THEN _AlarmNum := _CMD_Stop.ErrorID; END_IF
END_METHOD

METHOD PRIVATE M_UnlatchManuals
VAR_INPUT
END_VAR
VAR_INST
END_VAR
VAR_INST // added by the converter: edge detectors and wires of the graphical bodies
    _rt1, _rt2, _rt3, _rt4, _rt5 : R_TRIG;
END_VAR
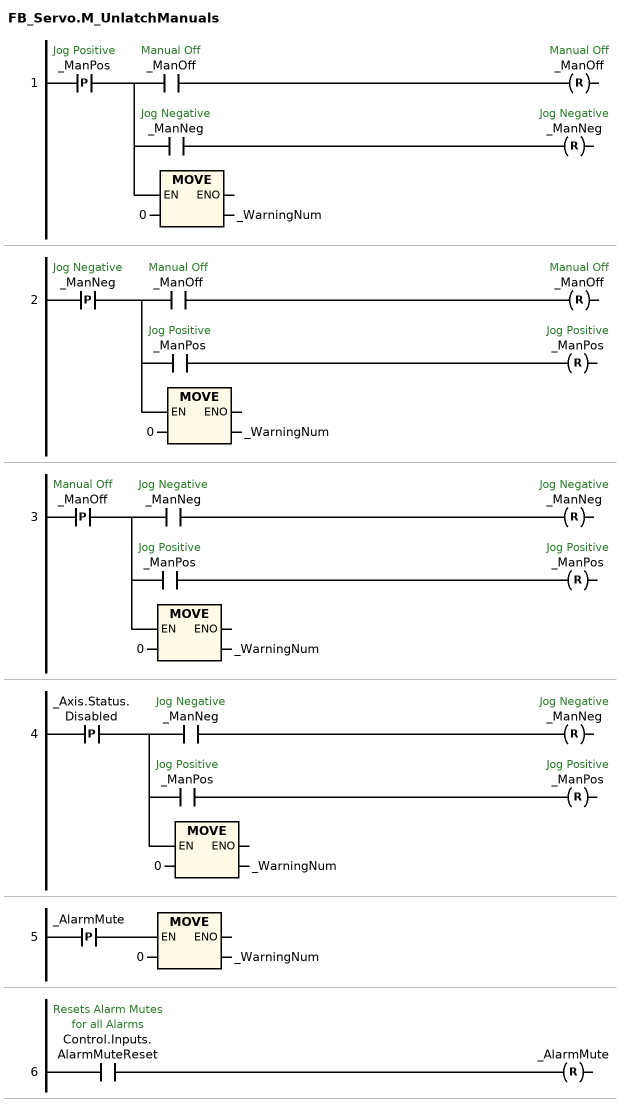
// NETWORK 1
//   _ManPos: Jog Positive
//   _ManOff: Manual Off
//   _ManNeg: Jog Negative
_rt1(CLK := _ManPos);
_ManOff R= _rt1.Q AND _ManOff;
_ManNeg R= _rt1.Q AND _ManNeg;
IF _rt1.Q THEN _WarningNum := 0; END_IF

// NETWORK 2
//   _ManNeg: Jog Negative
//   _ManOff: Manual Off
//   _ManPos: Jog Positive
_rt2(CLK := _ManNeg);
_ManOff R= _rt2.Q AND _ManOff;
_ManPos R= _rt2.Q AND _ManPos;
IF _rt2.Q THEN _WarningNum := 0; END_IF

// NETWORK 3
//   _ManOff: Manual Off
//   _ManNeg: Jog Negative
//   _ManPos: Jog Positive
_rt3(CLK := _ManOff);
_ManNeg R= _rt3.Q AND _ManNeg;
_ManPos R= _rt3.Q AND _ManPos;
IF _rt3.Q THEN _WarningNum := 0; END_IF

// NETWORK 4
//   _ManNeg: Jog Negative
//   _ManPos: Jog Positive
_rt4(CLK := _Axis.Status.Disabled);
_ManNeg R= _rt4.Q AND _ManNeg;
_ManPos R= _rt4.Q AND _ManPos;
IF _rt4.Q THEN _WarningNum := 0; END_IF

// NETWORK 5
_rt5(CLK := _AlarmMute);
IF _rt5.Q THEN _WarningNum := 0; END_IF

// NETWORK 6
//   Control.Inputs.AlarmMuteReset: Resets Alarm Mutes for all Alarms
_AlarmMute R= Control.Inputs.AlarmMuteReset;
END_METHOD

METHOD PRIVATE M_WarningMonitor
VAR_INPUT
END_VAR
VAR_INST
	{attribute 'tc_no_symbol'}                	                			
	_R_Trig				:   ARRAY[0..2] OF R_TRIG;
END_VAR
VAR_INST // added by the converter: edge detectors and wires of the graphical bodies
    _w1, _w2 : BOOL;
END_VAR
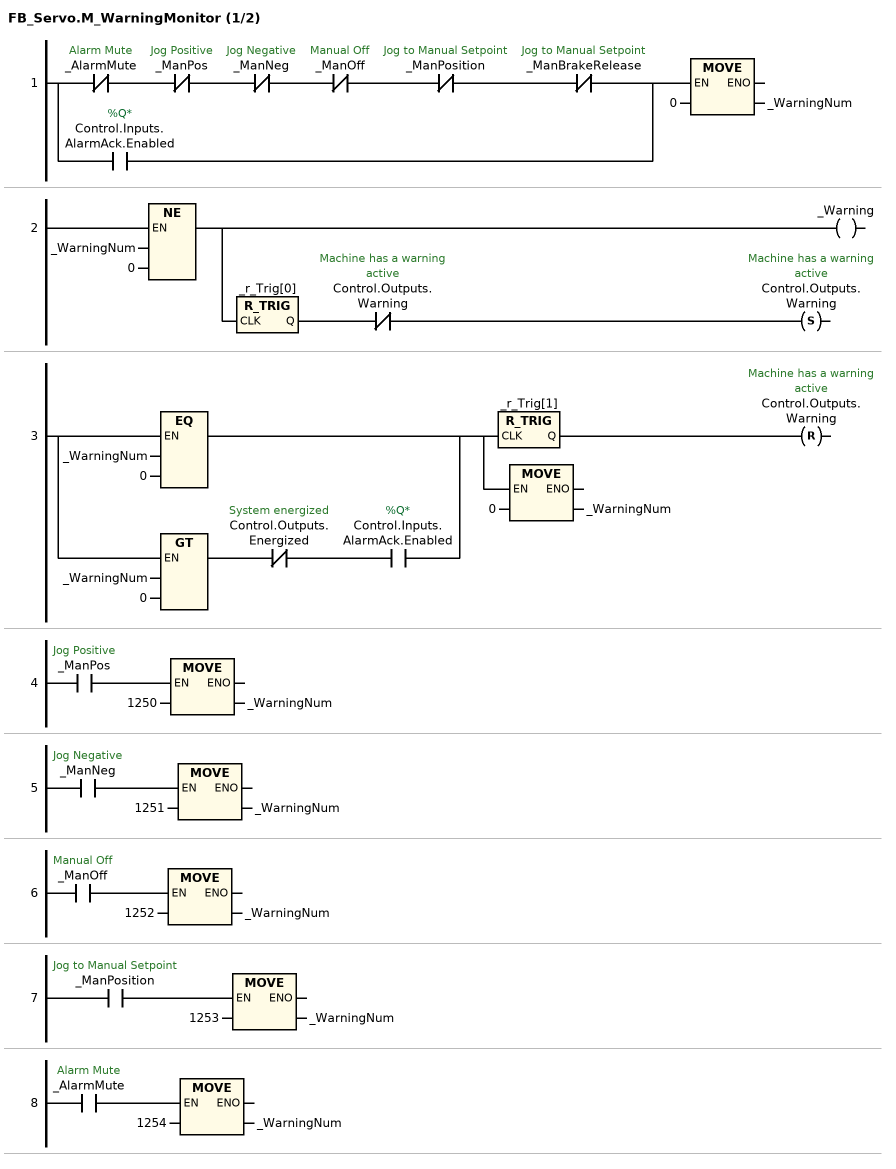
// NETWORK 1
//   _AlarmMute: Alarm Mute
//   _ManPos: Jog Positive
//   _ManNeg: Jog Negative
//   _ManOff: Manual Off
//   _ManPosition: Jog to Manual Setpoint
//   _ManBrakeRelease: Jog to Manual Setpoint
//   Control.Inputs.AlarmAck.Enabled: AT %Q*
IF NOT _AlarmMute AND NOT _ManPos AND NOT _ManNeg AND NOT _ManOff AND NOT _ManPosition AND NOT _ManBrakeRelease OR Control.Inputs.AlarmAck.Enabled THEN
    _WarningNum := 0;
END_IF

// NETWORK 2
//   Control.Outputs.Warning: Machine has a warning active
_w1 := _WarningNum <> 0;
_Warning := _w1;
_r_Trig[0](CLK := _w1); // R_TRIG
Control.Outputs.Warning S= _r_Trig[0].Q AND NOT Control.Outputs.Warning;

// NETWORK 3
//   Control.Outputs.Energized: System energized
//   Control.Inputs.AlarmAck.Enabled: AT %Q*
//   Control.Outputs.Warning: Machine has a warning active
_w2 := _WarningNum = 0 OR _WarningNum > 0 AND NOT Control.Outputs.Energized AND Control.Inputs.AlarmAck.Enabled;
_r_Trig[1](CLK := _w2); // R_TRIG
Control.Outputs.Warning R= _r_Trig[1].Q;
IF _w2 THEN _WarningNum := 0; END_IF

// NETWORK 4
//   _ManPos: Jog Positive
IF _ManPos THEN _WarningNum := 1250; END_IF

// NETWORK 5
//   _ManNeg: Jog Negative
IF _ManNeg THEN _WarningNum := 1251; END_IF

// NETWORK 6
//   _ManOff: Manual Off
IF _ManOff THEN _WarningNum := 1252; END_IF

// NETWORK 7
//   _ManPosition: Jog to Manual Setpoint
IF _ManPosition THEN _WarningNum := 1253; END_IF

// NETWORK 8
//   _AlarmMute: Alarm Mute
IF _AlarmMute THEN _WarningNum := 1254; END_IF

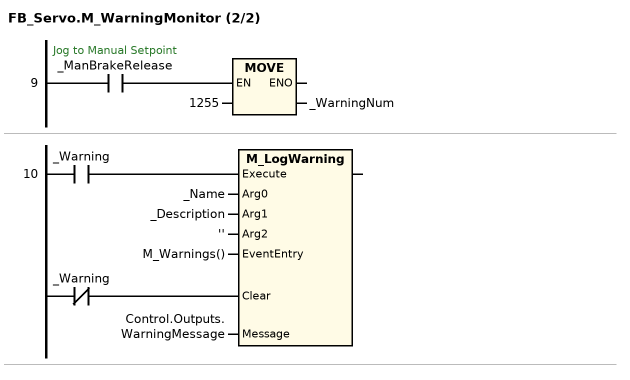
// NETWORK 9
//   _ManBrakeRelease: Jog to Manual Setpoint
IF _ManBrakeRelease THEN _WarningNum := 1255; END_IF

// NETWORK 10
M_LogWarning(Execute := _Warning, Arg0 := _Name, Arg1 := _Description, Arg2 := '', EventEntry := M_Warnings(), Clear := NOT _Warning, Message := Control.Outputs.WarningMessage);
END_METHOD

METHOD PRIVATE M_Warnings : TcEventEntry
VAR_INPUT
END_VAR
VAR_INST
END_VAR
CASE _WarningNum OF	
1150:    M_Warnings := 	TC_Events.TcServo.W_1150;			
1151:    M_Warnings :=  TC_Events.TcServo.W_1151;			
1152:    M_Warnings := 	TC_Events.TcServo.W_1152;			
1153:    M_Warnings := 	TC_Events.TcServo.W_1153;			
1154:    M_Warnings := 	TC_Events.TcServo.W_1154;	
1155:    M_Warnings :=  TC_Events.TcServo.W_1155;	
ELSE
		 M_Warnings := 	TC_Events.TcServo.W_Undefined;
END_CASE
END_METHOD

{attribute 'monitoring' := 'variable'}
PROPERTY PUBLIC ManBrakeRelease : Bool
SET
_ManBrakeRelease := ManBrakeRelease;
END_SET
END_PROPERTY

{attribute 'monitoring' := 'variable'}
PROPERTY PUBLIC ManEn : Bool
GET
ManEn := _ManEn;
END_GET
SET
_ManEn := ManEn;
END_SET
END_PROPERTY

{attribute 'monitoring' := 'variable'}
PROPERTY PUBLIC ManHome : REFERENCE TO ST_Selection
GET
ManHome REF= _ManHome;
END_GET
SET
_ManHome := ManHome;
END_SET
END_PROPERTY

{attribute 'monitoring' := 'variable'}
PROPERTY PUBLIC MoveDynamic : REFERENCE TO ARRAY[1..4] OF BOOL
GET
PUBLIC 
VAR
END_VAR
MoveDynamic REF= _MoveDynamic;
END_GET
SET
_MoveDynamic := MoveDynamic;
END_SET
END_PROPERTY

{attribute 'monitoring' := 'variable'}
PROPERTY PUBLIC MovePos : REFERENCE TO ARRAY[1..4] OF BOOL
GET
PUBLIC 
VAR
END_VAR
MovePos REF= _MovePos;
END_GET
SET
_MovePos := MovePos;
END_SET
END_PROPERTY

{attribute 'monitoring' := 'variable'}
PROPERTY PUBLIC MovePosSync : Bool
SET
_MovePosSync := MovePosSync;
END_SET
END_PROPERTY

{attribute 'monitoring' := 'variable'}
PROPERTY PUBLIC MoveSuperImpose : Bool
SET
_MoveSuperImpose := MoveSuperImpose;
END_SET
END_PROPERTY

{attribute 'monitoring' := 'variable'}
PROPERTY PUBLIC Moving : Bool
GET
Moving := _Moving;
END_GET
END_PROPERTY

{attribute 'monitoring' := 'variable'}
PROPERTY PUBLIC Name : String[15]
GET
Name := _Name;
END_GET
SET
_Name := Name;
END_SET
END_PROPERTY

{attribute 'monitoring' := 'variable'}
PROPERTY PUBLIC PosDynamicOK : REFERENCE TO ARRAY[1..4] OF BOOL
GET
PUBLIC 
VAR
END_VAR
PosDynamicOK REF= _PosDynamicOK;
END_GET
END_PROPERTY

{attribute 'Suspress_wrn_C0410'}
PROPERTY PUBLIC PosMove : REFERENCE TO ARRAY[1..4] OF ST_MovePosition_SP
GET
PUBLIC 
VAR
END_VAR
Posmove REF= _PosMove;
END_GET
SET
_Posmove := PosMove;
END_SET
END_PROPERTY

{attribute 'monitoring' := 'variable'}
PROPERTY PUBLIC PosMoveHome : REFERENCE TO ST_HomePosition_SP;
GET
PUBLIC 
VAR
END_VAR
PosMoveHome REF= _PosMoveHome;
END_GET
SET
_PosMoveHome := PosMoveHome;
END_SET
END_PROPERTY

{attribute 'monitoring' := 'variable'}
PROPERTY PUBLIC PosOK : REFERENCE TO ARRAY[1..4] OF BOOL
GET
PUBLIC 
VAR
END_VAR
PosOK REF= _PosOK;
END_GET
END_PROPERTY

{attribute 'monitoring' := 'variable'}
PROPERTY PUBLIC PosSyncOK : Bool
GET
PosSyncOK := _PosSyncOK;
END_GET
END_PROPERTY

{attribute 'monitoring' := 'variable'}
PROPERTY PUBLIC RunCam : Bool
SET
_RunCam := RunCam;
END_SET
END_PROPERTY

{attribute 'monitoring' := 'variable'}
PROPERTY PUBLIC StandStill : Bool
GET
StandStill := _StandStill;
END_GET
END_PROPERTY

{attribute 'monitoring' := 'variable'}
PROPERTY PUBLIC Unit : String[8]
GET
Unit := _Unit;
END_GET
SET
_Unit := Unit;
END_SET
END_PROPERTY

PROPERTY PUBLIC Variables : REFERENCE TO ARRAY[0..9] OF ST_Variable
GET
Variables REF= _Variables;
END_GET
END_PROPERTY

{attribute 'monitoring' := 'variable'}
PROPERTY PUBLIC Warning : Bool
GET
Warning := _Warning;
END_GET
END_PROPERTY

END_FUNCTION_BLOCK

// Objects/FB_Statistics_V4_02/FB_Statistics
FUNCTION_BLOCK FINAL FB_Statistics
VAR_INPUT
	Description				: STRING(31);			//Statistic description
	Trigger					: BOOL;					//New item trigger
	PerPulse				: REAL;					//Items per pulse
END_VAR
VAR
	_Reset					: BOOL;					//Reset Statistics
	_CycleTime				: REAL;					//Time for one item cycle (seconds)
	_CurrentRate			: REAL;					//Current item rate per minute
	_ThisMin				: REAL;					//Number of items processed this minute
	_LastMin				: REAL;					//Number of items processed last minute
	_ThisHour				: REAL;					//Number of items processed this hour
	_LastHour				: REAL;					//Number of items processed last hour
	_HistoryAvg				: REAL;					//Average items/minute for the previous 10 minutes
	_History				: ARRAY[1..10] OF REAL; //Item 10minute history
	_InstHistory			: ARRAY[1..20] OF REAL;	//Item instantaneous history
	_ItemCycleTime			: REAL;					//Item cycle time
	_InstHistoryCount		: INT;					//Instantaneous history For loop counter
	_HistoryCount			: INT;					//History For loop counter
	_HistorySum				: REAL;					//History summation holder
	_R_Trig					: R_TRIG;				//Statistic Count Trigger	
	_SecondsCount			: INT;					//Seconds history for loop counter
	_ThisSec				: INT;					//Item count this second
	_SecondsHistory			: ARRAY [0..59] OF INT; //Seconds history
	_ItemsLast60s			: INT;					//Current item rate for last 60 seconds
END_VAR
VAR_IN_OUT
	Control					: ST_System;			//Machine control system time
END_VAR
VAR PERSISTENT
	_LifeTime				: REAL;					//Life time count
	_Today					: REAL;					//Tadays count
END_VAR

//Statistic Count Trigger
_R_Trig	(CLK:=Trigger);

//Total Counts
IF Control.SystemTime.MidnightPulse OR _Reset THEN
	_Today := 0;
ELSE 
	IF _R_Trig.Q THEN
		_LifeTime := _LifeTime + PerPulse;
		_Today := _Today + PerPulse;
		_ThisHour := _ThisHour + PerPulse;
		_ThisMin := _ThisMin + PerPulse;
	END_IF
END_IF

//Cycle Time
IF _R_Trig.Q AND _ItemCycleTime > 0 THEN
	_CycleTime := _ItemCycleTime;
	_CurrentRate := PerPulse * (60 / F_CheckDivReal(_ItemCycleTime));
	_ItemCycleTime := 0;
	FOR _InstHistoryCount := 20 TO 2 BY -1 DO
		_InstHistory[F_CheckIndexBounds(1,10,_InstHistoryCount)] := _InstHistory[F_CheckIndexBounds(1,10,_InstHistoryCount)-1];
	END_FOR
	_InstHistory[1] := _CycleTime;	
ELSIF Control.PackMLState.Execute OR Control.PackMLState.Holding OR Control.PackMLState.UnHolding OR Control.PackMLState.Suspending OR Control.PackMLState.UnSuspending OR Control.PackMLState.Completing  THEN
	_ItemCycleTime := _ItemCycleTime + Control.SystemTime.ScanTime;
END_IF

//Minute Counts and History
IF Control.SystemTime.MinutePulse THEN
	_LastMin := _ThisMin;
	_ThisMin := 0;
	_HistorySum := 0;
	FOR _HistoryCount := 10 TO 2 BY -1 DO
		_History[F_CheckIndexBounds(1,10,_HistoryCount)] := _History[F_CheckIndexBounds(1,10,_HistoryCount)-1];
		_HistorySum := _HistorySum + _History[F_CheckIndexBounds(1,10,_HistoryCount)];
	END_FOR
	_History[1] := _LastMin;
	_HistorySum := _HistorySum + _History[1];
	_HistoryAvg := _HistorySum/10;
END_IF

//Hour counts
IF Control.SystemTime.HourPulse THEN
	_LastHour := _ThisHour;
	_ThisHour := 0;
END_IF

//Seconds Count and History
IF _R_Trig.Q THEN
	_SecondsHistory[_ThisSec] := _SecondsHistory[_ThisSec] + REAL_TO_INT(PerPulse);
END_IF

_ItemsLast60s := 0;
FOR _SecondsCount:= 0 TO 59 DO
	_ItemsLast60s := _ItemsLast60s + _SecondsHistory[_SecondsCount];
END_FOR

IF Control.SystemTime.SecondPulse THEN
	_ThisSec := _ThisSec + 1;
	IF _ThisSec >= 60 THEN _ThisSec := 0; END_IF;
	_SecondsHistory[_ThisSec] := 0;
END_IF

{attribute 'monitoring' := 'variable'}
PROPERTY PUBLIC CurrentRate : REAL
GET
CurrentRate := _CurrentRate;
END_GET
END_PROPERTY

{attribute 'monitoring' := 'variable'}
PROPERTY PUBLIC CycleTime : REAL
GET
CycleTime := _CycleTime;
END_GET
END_PROPERTY

{attribute 'monitoring' := 'variable'}
PROPERTY PUBLIC History : ARRAY[1..10] OF REAL
GET
History := _History;
END_GET
END_PROPERTY

{attribute 'monitoring' := 'variable'}
PROPERTY PUBLIC HistoryAvg : REAL
GET
HistoryAvg := _HistoryAvg;
END_GET
END_PROPERTY

{attribute 'monitoring' := 'variable'}
PROPERTY PUBLIC InstHistory : ARRAY[1..20] OF REAL
GET
InstHistory := _InstHistory;
END_GET
END_PROPERTY

{attribute 'monitoring' := 'variable'}
PROPERTY PUBLIC LastHour : REAL
GET
LastHour := _LastHour;
END_GET
END_PROPERTY

{attribute 'monitoring' := 'variable'}
PROPERTY PUBLIC LastMin : REAL
GET
PUBLIC 
VAR
END_VAR
LastMin := _LastMin;
END_GET
END_PROPERTY

{attribute 'monitoring' := 'variable'}
PROPERTY PUBLIC Reset : BOOL
GET
Reset := _Reset;
END_GET
SET
_Reset := Reset;
END_SET
END_PROPERTY

{attribute 'monitoring' := 'variable'}
PROPERTY PUBLIC ThisHour : REAL
GET
ThisHour := _ThisHour;
END_GET
END_PROPERTY

{attribute 'monitoring' := 'variable'}
PROPERTY PUBLIC ThisMin : REAL
GET
ThisMin := _ThisMin;
END_GET
END_PROPERTY

END_FUNCTION_BLOCK

// Objects/FB_StepEngine_V4_03/FB_StepEngine
FUNCTION_BLOCK FINAL FB_StepEngine EXTENDS FB_EventLogger  
VAR_INPUT
	Size					: UINT;
	Flags					: DWORD;
END_VAR             		
VAR_IN_OUT 
	Control					: ST_System;
	StepDesc				: ARRAY[*] OF STRING;
	MatrixA					: ARRAY[*] OF DINT;
	MatrixB					: ARRAY[*] OF DINT;
	MatrixC					: ARRAY[*] OF DINT;
	MatrixD					: ARRAY[*] OF DINT;
	TimerSP					: ARRAY[*] OF REAL;         		
END_VAR  
VAR_OUTPUT          		
	Outputs					: ARRAY[0..3] OF DINT; 
END_VAR             		
VAR      
	_StepReq				: INT;
	_DeviceAlarm			: BOOL;      		
	_SeqInterface			: ST_SequenceInterface;         		
	_StepTimeDn				: BOOL;
	_StepTimeRun			: BOOL;
	_StepChanged			: BOOL;
	_Disabled				: BOOL;
	_StepNum				: INT;
	_StepNumChan			: INT;
	_StepNumPrev			: INT;
	_StepTime_ET			: REAL;
	_StepTime_ETDT			: TIME;
	_StepTimeLeft			: REAL;
	_StepTimeLeftDT			: TIME;
	_StepTimePrev_ET		: REAL;
	_Message				: STRING;
	_Alarm					: BOOL;	
	_AlarmNum				: DINT;					
	_Fault					: BOOL;									
	_CurrentStep			: ARRAY[0..255] OF BOOL;
	_HistoryIndex			: INT;
END_VAR             		
VAR PERSISTENT      	
	_Name					: STRING[15];				
	_Description			: STRING[40];	
	_Disable				: BOOL;   			
	_AlarmMute				: BOOL;						
	_StepTime_PT			: REAL;
	_LastActiveStep			: INT;
	_History				: ARRAY[0..99] OF ST_SequenceHistory;	
	_Variables				: ARRAY [0..9] OF ST_Variable;									
END_VAR

M_AlarmMonitor();
F_CheckIndexBounds(0,UINT_TO_INT(Size),_StepNum);
F_CheckIndexBounds_REAL(0,65534,_StepTime_ET);
F_CheckIndexBounds_REAL(0,65534,_StepTime_PT);
F_CheckIndexBounds_REAL(0,65534,_StepTimeLeft);

IF  _Disable THEN
	_StepNum := 0;
	_Disabled := TRUE;
	_Message := 'Sequence Disabled';
ELSE
	_StepNum := _StepReq;
	_Disabled := FALSE;
	_Message:= StepDesc[_StepNum];
END_IF

IF Control.PackMLState.Complete THEN
	_LastActiveStep := 0;
END_IF

Outputs[0] := MatrixA[_StepNum];
Outputs[1] := MatrixB[_StepNum];
Outputs[2] := MatrixC[_StepNum];
Outputs[3] := MatrixD[_StepNum];

MEMSET(destAddr:= ADR(_CurrentStep), fillByte:= 0, n:= SIZEOF(_CurrentStep));
_CurrentStep[_StepNum] := TRUE;

IF _StepChanged THEN
	_StepTime_PT := TimerSP[_StepNum];
END_IF

_StepTime_ET := _StepTime_ET + Control.SystemTime.ScanTime;
_StepTime_ETDT := REAL_TO_TIME(_StepTime_ET);

IF _StepNum <> _StepNumChan THEN
	_StepTimePrev_ET := _StepTime_ET;
	_StepTime_ET := 0;
	_StepNumPrev := _StepNumChan;
	IF MatrixA[_StepNumChan].31 = TRUE THEN _LastActiveStep := _StepNumChan; END_IF
	IF MatrixA[_StepNumChan].30 = TRUE THEN _LastActiveStep := 0; END_IF	
	_StepNumChan := _StepNum;
	_StepChanged := TRUE;
	_StepTimeDn := FALSE;	
ELSE
	IF _StepTime_ET <= _StepTime_PT THEN
		_StepTimeLeft := _StepTime_PT - _StepTime_ET;
		_StepTimeLeftDT := REAL_TO_TIME(_StepTimeLeft);
	ELSE
		_StepTimeDn := TRUE;
	END_IF
	_StepChanged := FALSE;	
END_IF

IF _StepTime_PT = 0 THEN
	_StepTimeLeft := 0;
	_StepTimeLeftDT := REAL_TO_TIME(_StepTimeLeft);
END_IF

_History[0].StepNum:= _StepNum;
_History[0].StepTime:= _StepTime_ET;
_History[0].Message:= _Message;
	
IF _StepNumPrev <> _History[1].StepNum THEN 
	FOR _historyIndex:= 99 TO 2 BY -1 DO
		_History[F_CheckIndexBounds(0,99,_historyIndex)]:= _History[F_CheckIndexBounds(0,99,_historyIndex)-1];
	END_FOR
	_History[1].StepNum:= _StepNumPrev;
	_History[1].StepTime:= _StepTimePrev_ET;
	_History[1].Message:= StepDesc[_StepNumPrev];
END_IF

{attribute 'monitoring' := 'variable'}
PROPERTY PUBLIC Alarm : Bool
GET
Alarm := _Alarm;
END_GET
END_PROPERTY

{attribute 'monitoring' := 'variable'}
PROPERTY PUBLIC AlarmMute : BOOL
SET
AlarmMute := _AlarmMute;
END_SET
END_PROPERTY

{attribute 'monitoring' := 'variable'}
PROPERTY PUBLIC CurrentStep : REFERENCE TO ARRAY[0..255] OF BOOL
GET
CurrentStep REF= _CurrentStep;
END_GET
END_PROPERTY

{attribute 'monitoring' := 'variable'}
PROPERTY PUBLIC Description : String[40]
GET
Description := _Description;
END_GET
SET
_Description := Description;
END_SET
END_PROPERTY

{attribute 'monitoring' := 'variable'}
PROPERTY PUBLIC DeviceAlarm : BOOL
GET
DeviceAlarm :=_DeviceAlarm;
END_GET
SET
_DeviceAlarm := DeviceAlarm;
END_SET
END_PROPERTY

{attribute 'monitoring' := 'variable'}
PROPERTY PUBLIC Disable : BOOL
SET
_Disable := Disable;
END_SET
END_PROPERTY

{attribute 'monitoring' := 'variable'}
PROPERTY PUBLIC Disabled : BOOL
GET
PUBLIC 
VAR
END_VAR
Disabled := _Disabled;
END_GET
SET
_Disabled := Disabled;
END_SET
END_PROPERTY

{attribute 'monitoring' := 'variable'}
PROPERTY PUBLIC Fault : Bool
SET
_Fault := Fault;
END_SET
END_PROPERTY

PROPERTY PUBLIC History :REFERENCE to ARRAY[0..99] OF ST_SequenceHistory
GET
History REF=_History;
END_GET
END_PROPERTY

{attribute 'monitoring' := 'variable'}
PROPERTY PUBLIC LastActiveStep : int
GET
PUBLIC 
VAR
END_VAR
LastActiveStep := _LastActiveStep;
END_GET
SET
_LastActiveStep := LastActiveStep;
END_SET
END_PROPERTY

METHOD PROTECTED M_AlarmMonitor
VAR_INPUT
END_VAR
VAR_INST
END_VAR
VAR_INST // added by the converter: edge detectors and wires of the graphical bodies
    _w1, _w2 : BOOL;
END_VAR
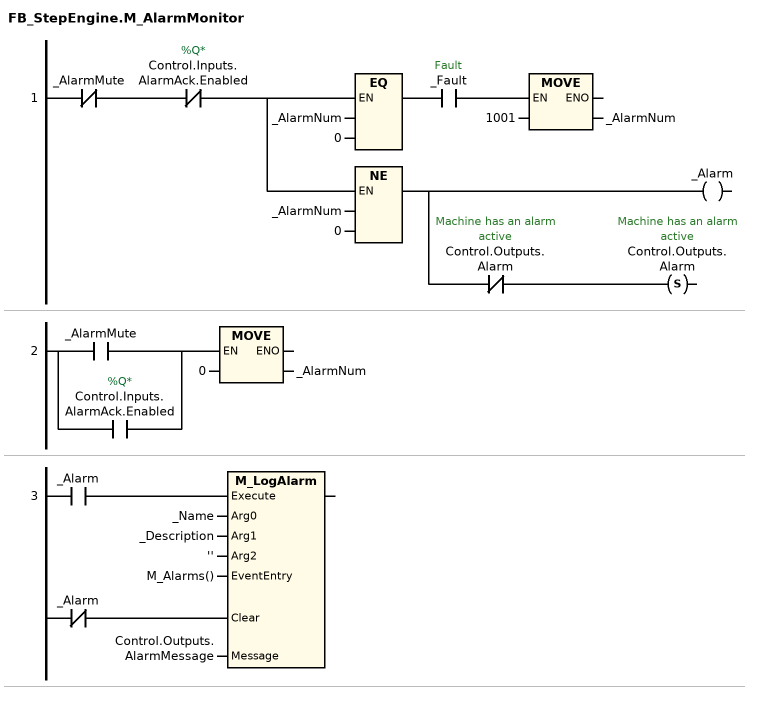
// NETWORK 1
//   Control.Inputs.AlarmAck.Enabled: AT %Q*
//   _Fault: Fault
//   Control.Outputs.Alarm: Machine has an alarm active
_w1 := NOT _AlarmMute AND NOT Control.Inputs.AlarmAck.Enabled;
IF (_w1 AND _AlarmNum = 0) AND _Fault THEN _AlarmNum := 1001; END_IF
_w2 := _w1 AND _AlarmNum <> 0;
_Alarm := _w2;
Control.Outputs.Alarm S= _w2 AND NOT Control.Outputs.Alarm;

// NETWORK 2
//   Control.Inputs.AlarmAck.Enabled: AT %Q*
IF _AlarmMute OR Control.Inputs.AlarmAck.Enabled THEN _AlarmNum := 0; END_IF

// NETWORK 3
M_LogAlarm(Execute := _Alarm, Arg0 := _Name, Arg1 := _Description, Arg2 := '', EventEntry := M_Alarms(), Clear := NOT _Alarm, Message := Control.Outputs.AlarmMessage);
END_METHOD

METHOD PRIVATE M_Alarms : TcEventEntry
VAR_INPUT
END_VAR
CASE _AlarmNum OF
	1001: M_Alarms:= TC_Events.TcSequence.A_1001;//Failed to Reach Requested State		
ELSE
	M_Alarms:= TC_Events.TcSequence.A_Undefined;
END_CASE
END_METHOD

{attribute 'monitoring' := 'variable'}
PROPERTY PUBLIC Name : String[15]
GET
Name := _Name;
END_GET
SET
_Name := Name;
END_SET
END_PROPERTY

{attribute 'monitoring' := 'variable'}
PROPERTY PUBLIC SeqInterface : REFERENCE TO ST_SequenceInterface
GET
SeqInterface REF= _SeqInterface;
END_GET
SET
_SeqInterface := SeqInterface;
END_SET
END_PROPERTY

{attribute 'monitoring' := 'variable'}
PROPERTY PUBLIC StepNum : INT
GET
PUBLIC 
VAR
END_VAR
StepNum := _StepNum;
END_GET
SET
PUBLIC 
VAR
END_VAR
_StepNum := StepNum;
END_SET
END_PROPERTY

{attribute 'monitoring' := 'variable'}
PROPERTY PUBLIC StepReq : INT
GET
StepReq := _StepReq;
END_GET
SET
_StepReq := StepReq;
END_SET
END_PROPERTY

{attribute 'monitoring' := 'variable'}
PROPERTY PUBLIC StepTime_ET : REAL
GET
PUBLIC 
VAR
END_VAR
StepTime_ET := _StepTime_ET;
END_GET
END_PROPERTY

{attribute 'monitoring' := 'variable'}
PROPERTY PUBLIC StepTimeDn : BOOL
GET
StepTimeDn := _StepTimeDn;
END_GET
END_PROPERTY

PROPERTY PUBLIC Variables : REFERENCE TO ARRAY[0..9] OF ST_Variable
GET
Variables REF= _Variables;
END_GET
END_PROPERTY

END_FUNCTION_BLOCK

// Objects/FB_TcpIpClient_V4_01/FB_TcpIpClient
FUNCTION_BLOCK FB_TcpIpClient EXTENDS FB_EventLogger 
VAR_INPUT
	Enable					: BOOL;//Enable TCP/IP Commnuication
	RemoteHost				: T_IPv4Addr := '127.0.0.1';//TCP/IP Socket IP Address
	RemotePort				: UDINT := 1024;//TCP/IP Socket Port
	ReconnectTime			: TIME := T#3S;//Time until reconnection is attempted
	AcceptPollingTime		: TIME := T#100MS;//Send poll time
	RecievePollingTime		: TIME := T#100MS;//Recieve poll Time
	RecieveTimeOut			: TIME := T#3S;// Recieve timeout
	TxData					: ANY;//Raw send data
	RxData					: ANY;//Raw recieve data
	Delimiter				: BYTE := 0;//String data type delimiter in ASCII format
END_VAR
VAR_IN_OUT
	Control					: ST_System;
END_VAR
VAR_OUTPUT
	Connected				: BOOL:= FALSE;//Established connection status
	SendRecieveRate			: REAL;//Time to send and recieve data over TCP/IP.
END_VAR
VAR
	{attribute 'tc_no_symbol'} 
	_fb_SocketConnect 		: FB_SocketConnect;		//Connects a Local client to a Remote Server
	{attribute 'tc_no_symbol'} 
	_fb_SocketClose			: FB_SocketClose;		//Closes an open TCP/IP socket. 
	{attribute 'tc_no_symbol'} 
	_fb_SocketSend			: FB_SocketSend;		//Sends data to a remote client or remote server via the TwinCAT TCP/IP Connection Server 
	{attribute 'tc_no_symbol'} 
	_fb_SocketReceive		: FB_SocketReceive;		//Data can be recieved from a remote client or remote server via the TwinCAT TCP/IP Connection Server 
	{attribute 'tc_no_symbol'} 
	_fb_ConnectTON			: TON;					//Reconnection Timer
	_eStep					: E_ConnectionSteps;	//TCPIP Connection Step
	_Alarm					: BOOL;					//Device Alarm
	_Warning				: BOOL;					//Device Warning
	_Message				: BOOL;					//Device Message
	_AlarmNum				: DINT;					//Device Alarm Number
	_WarningNum				: DINT;					//Device Warning Number
	_MessageNum				: DINT;					//Device Message Number
	_Fault					: BOOL;					//Device Fault
	_FaultTimer_ET			: REAL;					//Fault timer elapsed
	_ExtendedErrorCode		: UDINT;				//Extended Error Code
	_RecieveTimeOut			: BOOL;					//No bytes recieved in time error
	_RecieveBufferOverflow	: BOOL;					//No more free read buffer space error
	_r_Trig					: ARRAY[0..9] OF R_TRIG;//Public Rising Edge Triggers
END_VAR
VAR PERSISTENT
	_Name				: STRING[15];			//Name for HMI
	_Description		: STRING[40];			//Description for HMI
	_AlarmMute			: BOOL;					//Alarm Mute
	_FaultTimer_PT		: REAL;					//Fault timer preset time
END_VAR

M_AlarmMonitor();
M_WarningMonitor();
M_MessageMonitor();

IF Control.Inputs.AlarmMuteReset THEN _AlarmMute := FALSE; END_IF

CASE _eStep OF
	CONNECTION_STATE_IDLE:
		IF Enable XOR Connected THEN
			IF Enable THEN
				_fb_ConnectTON( IN := TRUE );
				IF _fb_ConnectTON.Q THEN
					_fb_ConnectTON( IN := FALSE, PT := ReconnectTime);
					_eStep := CONNECTION_STATE_CONNECT_START;
				END_IF
			ELSE
				_eStep := CONNECTION_STATE_CLOSE_START;
			END_IF
		ELSIF Connected THEN
			_eStep := CONNECTION_STATE_DATAEXCHANGE_START;
		ELSE
			_fb_ConnectTON( IN := FALSE, PT := T#0S );
		END_IF

	CONNECTION_STATE_CONNECT_START:
		_fb_SocketConnect( bExecute := FALSE );
		_fb_SocketConnect( sSrvNetID := '', sRemoteHost := RemoteHost, nRemotePort := RemotePort, bExecute := TRUE );
		_eStep := CONNECTION_STATE_CONNECT_WAIT;

	CONNECTION_STATE_CONNECT_WAIT:
		_fb_SocketConnect( bExecute := FALSE );
		IF NOT _fb_SocketConnect.bBusy THEN
			IF NOT _fb_SocketConnect.bError THEN
				Connected 	:= TRUE;
				_eStep := CONNECTION_STATE_IDLE;
			ELSE
				_eStep := CONNECTION_STATE_ERROR;
			END_IF
		END_IF
		
	CONNECTION_STATE_DATAEXCHANGE_START:
		M_DataExchange( Execute := FALSE,Socket := _fb_SocketConnect.hSocket);
		M_DataExchange( Execute := TRUE ,Socket :=_fb_SocketConnect.hSocket);
		_eStep := CONNECTION_STATE_DATAEXCHANGE_WAIT;

	CONNECTION_STATE_DATAEXCHANGE_WAIT:
		IF NOT M_DataExchange( Execute := FALSE,Socket := _fb_SocketConnect.hSocket) THEN
			_eStep := CONNECTION_STATE_IDLE;
		END_IF
		
	CONNECTION_STATE_CLOSE_START:
		_fb_SocketClose( bExecute := FALSE );
		_fb_SocketClose( sSrvNetID := '', hSocket:= _fb_SocketConnect.hSocket, bExecute:= TRUE );
		_eStep := CONNECTION_STATE_CLOSE_WAIT;

	CONNECTION_STATE_CLOSE_WAIT:
		_fb_SocketClose( bExecute := FALSE );
		IF NOT _fb_SocketClose.bBusy THEN
			Connected := FALSE;
			IF NOT _fb_SocketClose.bError THEN
				_eStep := CONNECTION_STATE_IDLE;
			ELSE
				_eStep := CONNECTION_STATE_ERROR;
			END_IF
		END_IF

	CONNECTION_STATE_ERROR:(* Error step *)
		IF Connected THEN
			_eStep := CONNECTION_STATE_CLOSE_START;
		ELSE
			_eStep := CONNECTION_STATE_IDLE;
		END_IF
END_CASE

{attribute 'monitoring' := 'variable'}
PROPERTY PUBLIC Alarm : Bool
GET
Alarm := _Alarm;
END_GET
END_PROPERTY

{attribute 'monitoring' := 'variable'}
PROPERTY PUBLIC AlarmMute : BOOL
SET
AlarmMute := _AlarmMute;
END_SET
END_PROPERTY

{attribute 'monitoring' := 'variable'}
PROPERTY PUBLIC Description : String[40]
GET
Description := _Description;
END_GET
SET
_Description := Description;
END_SET
END_PROPERTY

{attribute 'monitoring' := 'variable'}
PROPERTY PUBLIC Fault : Bool
SET
_Fault := Fault;
END_SET
END_PROPERTY

{attribute 'monitoring' := 'variable'}
PROPERTY PUBLIC FaultTimer_PT : real
GET
FaultTimer_PT := _FaultTimer_PT;
END_GET
SET
_FaultTimer_PT := FaultTimer_PT;
END_SET
END_PROPERTY

METHOD PRIVATE M_AlarmMonitor
VAR_INPUT
END_VAR
VAR_INST
END_VAR
VAR_INST // added by the converter: edge detectors and wires of the graphical bodies
    _w1, _w2, _w3, _w4, _w5 : BOOL;
    _rt1, _rt2, _rt3, _rt4, _rt5, _rt6 : R_TRIG;
END_VAR
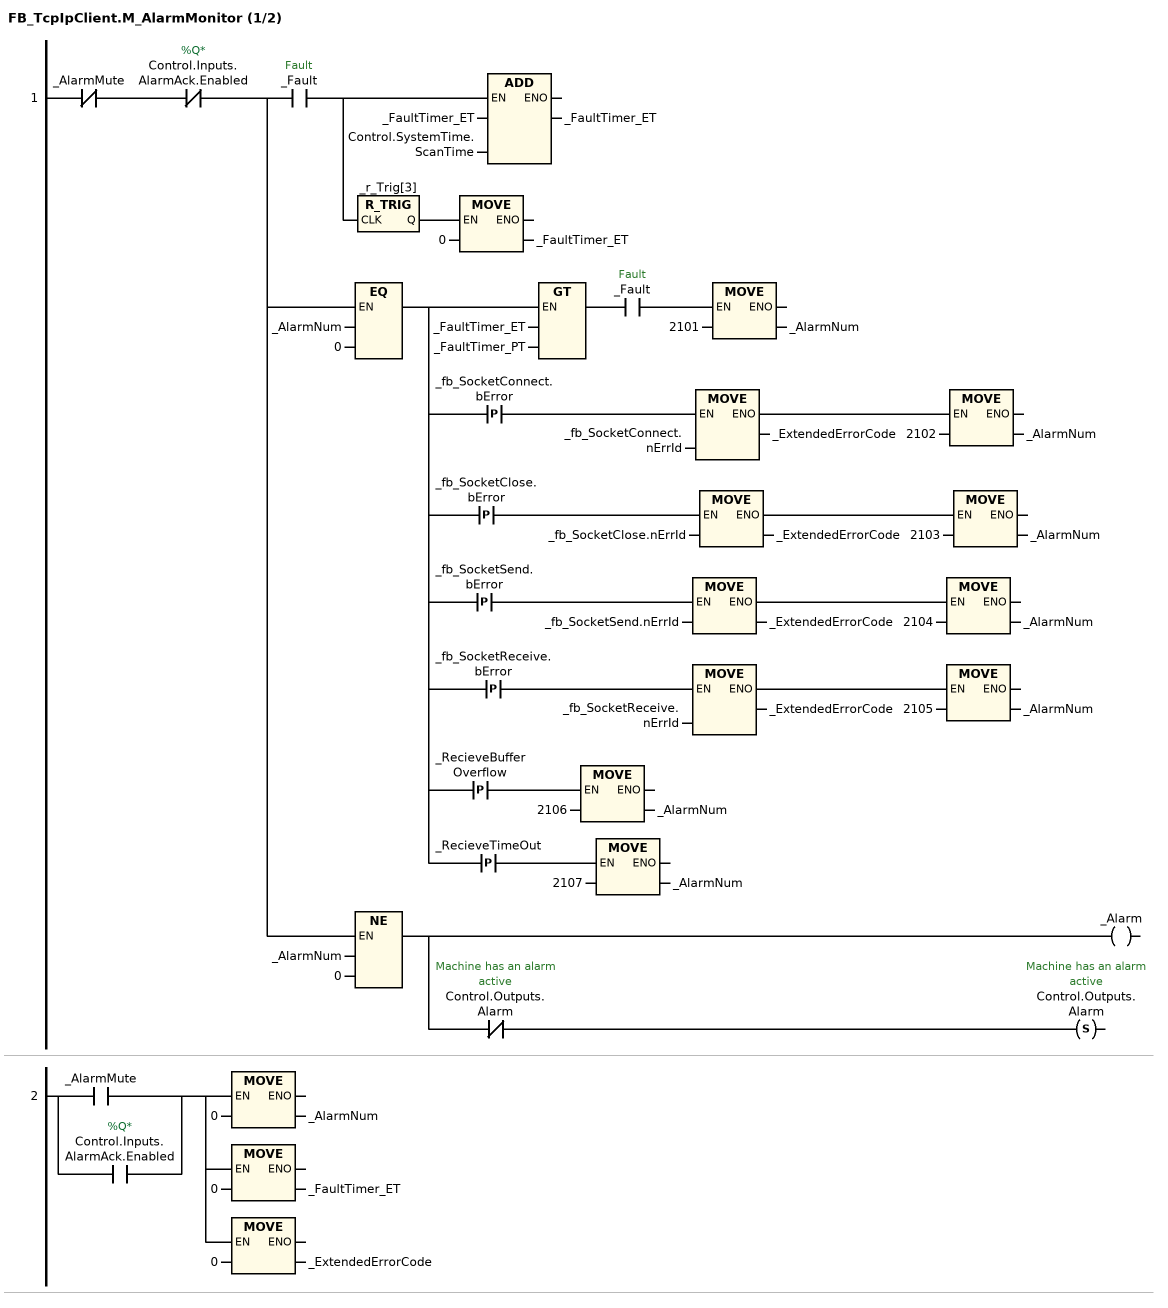
// NETWORK 1
//   Control.Inputs.AlarmAck.Enabled: AT %Q*
//   _Fault: Fault
//   _FaultTimer_ET: Fault timer elapsed
//   Control.SystemTime.ScanTime: Last scan time (Seconds)
//   _FaultTimer_PT: Fault timer preset time
//   Control.Outputs.Alarm: Machine has an alarm active
_w1 := NOT _AlarmMute AND NOT Control.Inputs.AlarmAck.Enabled;
_w2 := _w1 AND _Fault;
IF _w2 THEN _FaultTimer_ET := _FaultTimer_ET + Control.SystemTime.ScanTime; END_IF
_r_Trig[3](CLK := _w2); // R_TRIG
IF _r_Trig[3].Q THEN _FaultTimer_ET := 0; END_IF
_w3 := _w1 AND _AlarmNum = 0;
IF (_w3 AND _FaultTimer_ET > _FaultTimer_PT) AND _Fault THEN _AlarmNum := 2101; END_IF
_rt1(CLK := _fb_SocketConnect.bError);
IF _w3 AND _rt1.Q THEN _ExtendedErrorCode := _fb_SocketConnect.nErrId; END_IF
IF _w3 AND _rt1.Q THEN _AlarmNum := 2102; END_IF
_rt2(CLK := _fb_SocketClose.bError);
IF _w3 AND _rt2.Q THEN _ExtendedErrorCode := _fb_SocketClose.nErrId; END_IF
IF _w3 AND _rt2.Q THEN _AlarmNum := 2103; END_IF
_rt3(CLK := _fb_SocketSend.bError);
IF _w3 AND _rt3.Q THEN _ExtendedErrorCode := _fb_SocketSend.nErrId; END_IF
IF _w3 AND _rt3.Q THEN _AlarmNum := 2104; END_IF
_rt4(CLK := _fb_SocketReceive.bError);
IF _w3 AND _rt4.Q THEN _ExtendedErrorCode := _fb_SocketReceive.nErrId; END_IF
IF _w3 AND _rt4.Q THEN _AlarmNum := 2105; END_IF
_rt5(CLK := _RecieveBufferOverflow);
IF _w3 AND _rt5.Q THEN _AlarmNum := 2106; END_IF
_rt6(CLK := _RecieveTimeOut);
IF _w3 AND _rt6.Q THEN _AlarmNum := 2107; END_IF
_w4 := _w1 AND _AlarmNum <> 0;
_Alarm := _w4;
Control.Outputs.Alarm S= _w4 AND NOT Control.Outputs.Alarm;

// NETWORK 2
//   Control.Inputs.AlarmAck.Enabled: AT %Q*
//   _FaultTimer_ET: Fault timer elapsed
_w5 := _AlarmMute OR Control.Inputs.AlarmAck.Enabled;
IF _w5 THEN _AlarmNum := 0; END_IF
IF _w5 THEN _FaultTimer_ET := 0; END_IF
IF _w5 THEN _ExtendedErrorCode := 0; END_IF

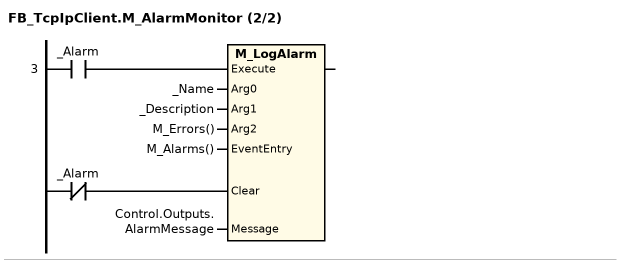
// NETWORK 3
M_LogAlarm(Execute := _Alarm, Arg0 := _Name, Arg1 := _Description, Arg2 := M_Errors(), EventEntry := M_Alarms(), Clear := NOT _Alarm, Message := Control.Outputs.AlarmMessage);
END_METHOD

METHOD M_Alarms : TcEventEntry
VAR_INPUT
END_VAR
CASE _AlarmNum OF
	2101: M_Alarms:= TC_Events.TcTcpIpClient.A_2101;//General error	
	2102: M_Alarms:= TC_Events.TcTcpIpClient.A_2102;//Socket connection error	
	2103: M_Alarms:= TC_Events.TcTcpIpClient.A_2103;//Socket close error	
	2104: M_Alarms:= TC_Events.TcTcpIpClient.A_2104;//Socket send error		
	2105: M_Alarms:= TC_Events.TcTcpIpClient.A_2105;//Socket recieve error		
	2106: M_Alarms:= TC_Events.TcTcpIpClient.A_2106;//Receive buffer overflow	
	2107: M_Alarms:= TC_Events.TcTcpIpClient.A_2107;//Receive timeout error				
ELSE
	M_Alarms:= TC_Events.TcTcpIpClient.A_Undefined;
END_CASE
END_METHOD

METHOD PRIVATE M_DataExchange : BOOL;
VAR_INPUT
	Socket				: T_HSOCKET;
	Execute				: BOOL;
END_VAR             	
VAR_INST
	{attribute 'tc_no_symbol'} 
	_Busy				: BOOL;
	{attribute 'tc_no_symbol'} 
	_Error 				: BOOL;
	{attribute 'tc_no_symbol'} 
	_eStep				: E_ClientDataExchangeSteps;
	{attribute 'tc_no_symbol'} 
	_fb_ReceiveTON		: TON;
	{attribute 'tc_no_symbol'} 
	_fb_DisconnectTON 	: TON;
	{attribute 'tc_no_symbol'} 
	_cbFrame			: UDINT;
	{attribute 'tc_no_symbol'} 
	_rxBuffer			: ARRAY[0..255] OF BYTE;
	{attribute 'tc_no_symbol'} 
	_SendRecieveRate	: REAL;
	{attribute 'tc_no_symbol'} 
	_cbReceived, _startPos, _endPos, _idx	: UDINT;
END_VAR
_r_Trig[9]( CLK := Execute );
IF _SendRecieveRate > SendRecieveRate THEN SendRecieveRate :=  _SendRecieveRate; END_IF
_SendRecieveRate := _SendRecieveRate + Control.SystemTime.ScanTime;
CASE _eStep OF

	CLIENT_DATAEXCHANGE_STATE_IDLE:
		IF _r_Trig[9].Q THEN
			_SendRecieveRate := 0;
			_Busy 	:= TRUE;
			_Error 	:= FALSE;
			_fb_DisconnectTON( IN := FALSE, PT := T#0MS );(* disable timeout check first *)
			_fb_ReceiveTON( IN := FALSE, PT := T#0MS ); (* receive first request immediately *)
			_eStep 	:= CLIENT_DATAEXCHANGE_STATE_SEND_START;
		END_IF
		
	CLIENT_DATAEXCHANGE_STATE_SEND_START:
		_fb_SocketSend( bExecute := FALSE );
		_fb_SocketSend(	hSocket	:= Socket ,pSrc	:= TxData.pValue,cbLen:=DINT_TO_UDINT(TxData.diSize),bExecute:= TRUE );
		_eStep := CLIENT_DATAEXCHANGE_STATE_SEND_WAIT;

	CLIENT_DATAEXCHANGE_STATE_SEND_WAIT:
		_fb_SocketSend( bExecute := FALSE );
		IF NOT _fb_SocketSend.bBusy THEN
			IF NOT _fb_SocketSend.bError THEN
				_eStep := CLIENT_DATAEXCHANGE_STATE_RECEIVE_START;
			ELSE
				_eStep := CLIENT_DATAEXCHANGE_STATE_ERROR;
			END_IF
		END_IF

	CLIENT_DATAEXCHANGE_STATE_RECEIVE_START: (* Receive remote client data *)
		_fb_ReceiveTON(  IN := TRUE );
		IF _fb_ReceiveTON.Q THEN
			_fb_ReceiveTON( IN := FALSE );
			_fb_SocketReceive( bExecute := FALSE );
			MEMSET(ADR( _rxBuffer ),0,SIZEOF( _rxBuffer ));
			IF RxData.TypeClass = DINT_TO_UDINT(IBaseLibrary.TYPE_STRING) THEN
				_fb_SocketReceive( hSocket:= Socket,pDest:= ADR( _rxBuffer ), cbLen:= SIZEOF( _rxBuffer ),bExecute:= TRUE );
			ELSE
				_fb_SocketReceive( hSocket:= Socket,pDest := RxData.pValue, cbLen:=DINT_TO_UDINT(RxData.diSize),bExecute:= TRUE );
			END_IF
			_eStep := CLIENT_DATAEXCHANGE_STATE_RECEIVE_WAIT;
		END_IF

	CLIENT_DATAEXCHANGE_STATE_RECEIVE_WAIT:
		_fb_SocketReceive( bExecute := FALSE );
		IF NOT _fb_SocketReceive.bBusy THEN
			IF NOT _fb_SocketReceive.bError THEN
				IF (_fb_SocketReceive.nRecBytes > 0) THEN(* bytes received *)
					IF RxData.TypeClass = DINT_TO_UDINT(IBaseLibrary.TYPE_STRING) THEN
						_startPos 	:= _cbReceived;(* rxBuffer array index of first data byte *)
						_endPos  	:= _cbReceived + _fb_SocketReceive.nRecBytes  - 1;(* rxBuffer array index of last data byte *)
						_cbReceived 	:= _cbReceived + _fb_SocketReceive.nRecBytes;(* calculate the number of received data bytes *)
						_cbFrame	:= 0;(* reset frame length *)
                	
						IF _cbReceived < DINT_TO_UDINT(RxData.diSize) THEN (* no overflow *)
                	
							_fb_ReceiveTON( IN := FALSE, PT := T#0S ); (* bytes received => increase the read (polling) speed *)
							_fb_DisconnectTON( IN := FALSE, PT := RecieveTimeOut);(* bytes received => disable timeout check *)
                	
							(* search for string end delimiter *)
							FOR _idx := _startPos TO _endPos BY 1 DO
								IF _rxBuffer[_idx] = Delimiter THEN(* string end delimiter found *)
									_cbFrame := _idx + 1;(* calculate the length of the received string (inclusive the end delimiter) *)
									MEMCPY(  RxData.pValue, ADR( _rxBuffer ), _cbFrame );(* copy the received string to the output variable (inclusive the end delimiter) *)
									MEMMOVE( ADR( _rxBuffer ), ADR( _rxBuffer[_cbFrame] ),  _cbReceived - _cbFrame  );(* move the reamaining data bytes *)
									_cbReceived := _cbReceived - _cbFrame;(* recalculate the reamaining data byte length *)
									_Busy := FALSE;
									_eStep := CLIENT_DATAEXCHANGE_STATE_IDLE;
									EXIT;
								END_IF
							END_FOR
                	
						ELSE(* there is no more free read buffer space => the answer string should be terminated *)
							_RecieveBufferOverflow := TRUE;
							_eStep := CLIENT_DATAEXCHANGE_STATE_ERROR;
						END_IF
					ELSE
						_Busy := FALSE;
						_eStep := CLIENT_DATAEXCHANGE_STATE_IDLE;
					END_IF

				ELSE(* no bytes received *)
					_fb_ReceiveTON( IN := FALSE, PT := RecievePollingTime);(* no bytes received => decrease the read (polling) speed *)
					_fb_DisconnectTON( IN := TRUE, PT := RecieveTimeOut );(* no bytes received => enable timeout check*)
					IF _fb_DisconnectTON.Q THEN (* timeout error*)
						_fb_DisconnectTON( IN := FALSE );
						_RecieveTimeOut:= TRUE;
						_eStep := CLIENT_DATAEXCHANGE_STATE_ERROR;
					ELSE(* repeat reading *)
						_eStep := CLIENT_DATAEXCHANGE_STATE_RECEIVE_START; (* repeat reading *)
					END_IF
				END_IF
			ELSE(* receive error *)
				_eStep := CLIENT_DATAEXCHANGE_STATE_ERROR;
			END_IF
		END_IF

	CLIENT_DATAEXCHANGE_STATE_ERROR:
		_Busy := FALSE;
		_RecieveTimeOut:= FALSE;
		_RecieveBufferOverflow := FALSE;
		_Error := TRUE;
		_SendRecieveRate := 0;
		_cbReceived := 0;
		_eStep := CLIENT_DATAEXCHANGE_STATE_IDLE;
END_CASE

M_DataExchange:= _Busy;
END_METHOD

METHOD PRIVATE M_Errors : STRING(126)
VAR_INPUT
END_VAR
VAR_INST
END_VAR
CASE _ExtendedErrorCode OF	
//Global Error Codes
0	: M_Errors :='';
1	: M_Errors :='1 Internal error';	 	 
2	: M_Errors :='2 No Rtime';	 	 
3	: M_Errors :='3	Allocation locked memory error';	 	 
4	: M_Errors :='4	Insert mailbox error';
5	: M_Errors :='5	Wrong receive HMSG';	 	 
6	: M_Errors :='6	target port not found	ADS Server not started';	 
7	: M_Errors :='7	target machine not found Missing ADS routes';	 
8	: M_Errors :='8	Unknown command ID';	 	 
9	: M_Errors :='9	Bad task ID';	 	 
10	: M_Errors :='10 No IO';	 	 
11	: M_Errors :='11 Unknown ADS command';	 	 
12	: M_Errors :='12 Win 32 error';	 	 
13	: M_Errors :='13 Port not connected';	 	 
14	: M_Errors :='14 Invalid ADS length';	 	 
15	: M_Errors :='15 Invalid AMS Net ID';	 	 
16	: M_Errors :='16 Low Installation level';	 	 
17	: M_Errors :='17 No debug available';	 	 
18	: M_Errors :='18 Port disabled';	 	 
19	: M_Errors :='19 Port already connected';	 	 
20	: M_Errors :='20 ADS Sync Win32 error';	 	 
21	: M_Errors :='21 ADS Sync Timeout';	 	 
22	: M_Errors :='22 ADS Sync AMS error';	 	 
23	: M_Errors :='23 ADS Sync no index map';	 	 
24	: M_Errors :='24 Invalid ADS port';	 	 
25	: M_Errors :='25 No memory';	 	 
26	: M_Errors :='26 TCP send error';	 	 
27	: M_Errors :='27 Host unreachable'; 	 
28	: M_Errors :='28 Invalid AMS fragment';
//Router Error Codes
1280 :	M_Errors :='1280 No locked memory can be allocated'; 
1281 :	M_Errors :='1281 The size of the router memory could not be changed'; 	 
1282 :	M_Errors :='1282 The mailbox has reached the maximum number OF possible messages'; 
1283 :	M_Errors :='1283 The mailbox has reached the maximum number OF possible messages'; 
1284 :	M_Errors :='1284 The port type is unknown'; 	 
1285 :	M_Errors :='1285 Router is not initialised'; 	 
1286 :	M_Errors :='1286 The desired port number is already assigned'; 	 
1287 :	M_Errors :='1287 Port not registered'; 	 
1288 :	M_Errors :='1288 The maximum number of Ports reached'; 	 
1289 :	M_Errors :='1289 The port is invalid'; 	 
1290 :	M_Errors :='1290 TwinCAT Router not active';  
1291 :	M_Errors :='1291 ROUTERERR_FRAGMENTBOXFULL'; 	 	 
1292 :	M_Errors :='1292 ROUTERERR_FRAGMENTTIMEOUT'; 	 	 
1293 :	M_Errors :='1293 ROUTERERR_TOBEREMOVED'; 
//General ADS Error Codes
1792: M_Errors :='1792 error class <device error>';	 	 
1793: M_Errors :='1793 Service is not supported by server';	 	 
1794: M_Errors :='1794 invalid index group';	 	 
1795: M_Errors :='1795 invalid index offset';	 	 
1796: M_Errors :='1796 reading/writing not permitted';	 	 
1797: M_Errors :='1797 parameter size not correct';	 	 
1798: M_Errors :='1798 invalid parameter value(S)';	 	 
1799: M_Errors :='1799 device is not in a ready state';	 	 
1800: M_Errors :='1800 device is busy';	 	 
1801: M_Errors :='1801 invalid context (must be in Windows)';	 	 
1802: M_Errors :='1802 out OF memory';	 	 
1803: M_Errors :='1803 invalid parameter value(s)';	 	 
1804: M_Errors :='1804 not found (files, ...)';	 	 
1805: M_Errors :='1805 syntax error in command or file';	 	 
1806: M_Errors :='1806 objects DO not match';	 	 
1807: M_Errors :='1807 object already exists';	 	 
1808: M_Errors :='1808 symbol not found';	 	 
1809: M_Errors :='1809 symbol version invalid';	
1810: M_Errors :='1810 server is in invalid state';	 	 
1811: M_Errors :='1811 AdsTransMode not supported';	 	 
1812: M_Errors :='1812 notification handle is invalid';	
1813: M_Errors :='1813 notification client not registered';	 	 
1814: M_Errors :='1814 no more notification handles';	 	 
1815: M_Errors :='1815 size for watch too big';	 	 
1816: M_Errors :='1816 device not initialized';	 	 
1817: M_Errors :='1817 device has a timeout';	 	 
1818: M_Errors :='1818 query INTERFACE failed';	 	 
1819: M_Errors :='1819 wrong interface required';	 	 
1820: M_Errors :='1820 class ID is invalid';	 	 
1821: M_Errors :='1821 object ID is invalid';	 	 
1822: M_Errors :='1822 request is pending';	 	 
1823: M_Errors :='1823 request is aborted';	 	 
1824: M_Errors :='1824 signal warning';	 	 
1825: M_Errors :='1825 invalid array index';	 	 
1826: M_Errors :='1826 symbol not active';	
1827: M_Errors :='1827 access denied';	 	 
1828: M_Errors :='1828 missing license';	 	
1836: M_Errors :='1836 exception occured during system start';	
1856: M_Errors :='1856 Error class <client error>';	 	 
1857: M_Errors :='1857 invalid parameter at service';	 	 
1858: M_Errors :='1858 polling list is empty';	 	 
1859: M_Errors :='1859 var connection already in use';	 	 
1860: M_Errors :='1860 invoke ID in use';	 	 
1861: M_Errors :='1861 timeout elapsed'; 	
1862: M_Errors :='1862 error in win32 subsystem';	 	 
1863: M_Errors :='1863 Invalid client timeout value';	 	 
1864: M_Errors :='1864 ads-port not opened';	 	 
1872: M_Errors :='1872 internal error in ads sync';	 	 
1873: M_Errors :='1873 hash table overflow';	 	 
1874: M_Errors :='1874 key not found in hash';	 	 
1875: M_Errors :='1875 no more symbols in cache';	 	 
1876: M_Errors :='1876 invalid response received';	 	 
1877: M_Errors :='1877 sync port is locked';
//RTime Error Codes
4096: M_Errors:= '4096 INTERNAL error in the REAL-TIME system.';
4097: M_Errors:= '4097 Timer value is NOT valid.';
4098: M_Errors:= '4098 Task pointer has the invalid value 0 (zero).';
4099: M_Errors:= '4099 Stack POINTER has the invalid value 0 (zero).';
4100: M_Errors:= '4100 The request task priority is already assigned.';
4101: M_Errors:= '4101 No free TCB (Task Control Block) available. The maximum number OF TCBs is 64.';
4102: M_Errors:= '4102 No free semaphores available. The maximum number of semaphores is 64.';
4103: M_Errors:= '4103 No free space available in the queue. The maximum number OF positions in the queue is 64.';
4109: M_Errors:= '4109 An external synchronization interrupt is already applied.';
4110: M_Errors:= '4110 No external sync interrupt applied.';
4111: M_Errors:= '4111 Application of the external synchronization interrupt has failed.';
4112: M_Errors:= '4112 Call OF a service FUNCTION in the wrong context';
4119: M_Errors:= '4119 Intel VT-x extension is not supported.';
4120: M_Errors:= '4120 Intel VT-x extension is NOT enabled in the BIOS.';
4121: M_Errors:= '4121 Missing function in Intel VT-x extension.';
4122: M_Errors:= '4122 Activation OF Intel VT-x fails.';
//TCP Winsock Error Codes
10060: M_Errors:= '10060 Intel VT-x extension is NOT enabled in the BIOS.';
10061: M_Errors:= '10061 Missing function in Intel VT-x extension.';
10065: M_Errors:= '10065 Activation OF Intel VT-x fails.';
//Internal error codes of the TwinCAT TCP/IP Connection Server
32769: M_Errors:= '32769 No new sockets can be created (for FB_SocketListen AND FB_SocketConnect).';
32770: M_Errors:= '32770 Socket handle is invalid (for FB_SocketReceive, FB_SocketAccept, FB_SocketSend etc.).';
32771: M_Errors:= '32771 Is returned when FB_SocketListen is called, if the TcpIp port listener already exists.';
32772: M_Errors:= '32772 Is returned when FB_SocketReceive is called, if the client socket is no longer connected with the server.';
32773: M_Errors:= '32773 Is returned when FB_SocketAccept is called, if an error was registered in the listener socket.';
//Internal SNMP error codes
36865: M_Errors:= '36865 INCORRECT PARAMETER SIZE';
36866: M_Errors:= '36866 INVALID PARAMETER';
ELSE
	M_Errors := 	CONCAT('Undefined TCP Server Error - ' , TO_STRING( _ExtendedErrorCode));
END_CASE
END_METHOD

METHOD PRIVATE M_MessageMonitor
VAR_INPUT
END_VAR
VAR_INST
END_VAR
VAR_INST // added by the converter: edge detectors and wires of the graphical bodies
    _w1 : BOOL;
    _rt1 : R_TRIG;
    _ft1 : F_TRIG;
END_VAR
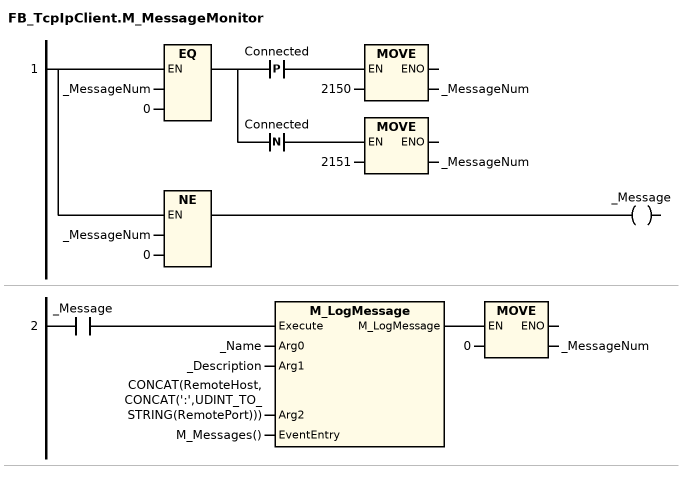
// NETWORK 1
_w1 := _MessageNum = 0;
_rt1(CLK := Connected);
IF _w1 AND _rt1.Q THEN _MessageNum := 2150; END_IF
_ft1(CLK := Connected);
IF _w1 AND _ft1.Q THEN _MessageNum := 2151; END_IF
_Message := _MessageNum <> 0;

// NETWORK 2
IF M_LogMessage(Execute := _Message, Arg0 := _Name, Arg1 := _Description, Arg2 := CONCAT(RemoteHost,CONCAT(':',UDINT_TO_STRING(RemotePort))), EventEntry := M_Messages()) THEN
    _MessageNum := 0;
END_IF
END_METHOD

METHOD PRIVATE M_Messages : TcEventEntry
VAR_INPUT
END_VAR
CASE _MessageNum OF
	2150: M_Messages:= TC_Events.TcTcpIpClient.M_2150;//Socket connection open
	2151: M_Messages:= TC_Events.TcTcpIpClient.M_2151;//Socket connection closed
END_CASE
END_METHOD

METHOD PRIVATE M_WarningMonitor
VAR_INPUT
END_VAR
VAR_INST
END_VAR
VAR_INST // added by the converter: edge detectors and wires of the graphical bodies
    _w1 : BOOL;
END_VAR
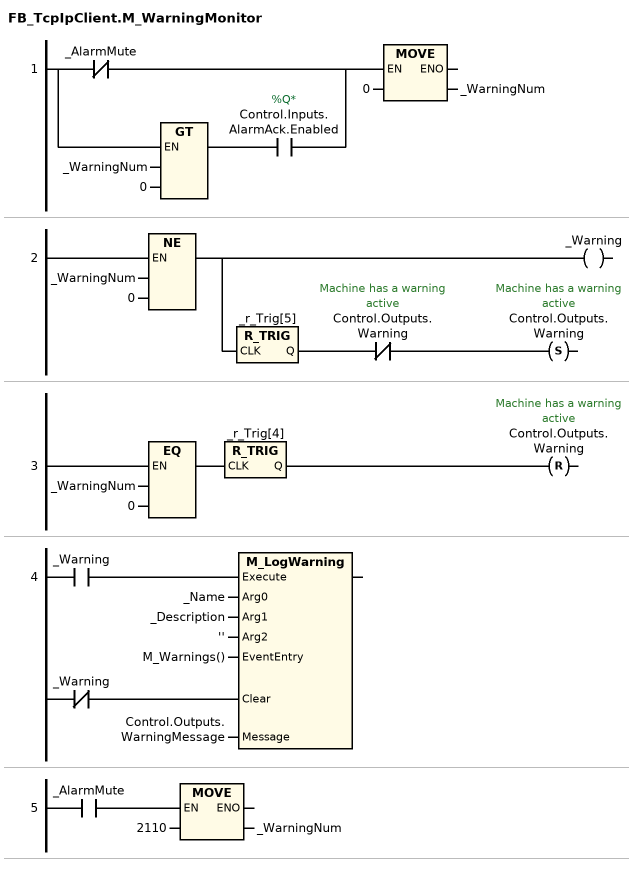
// NETWORK 1
//   Control.Inputs.AlarmAck.Enabled: AT %Q*
IF NOT _AlarmMute OR _WarningNum > 0 AND Control.Inputs.AlarmAck.Enabled THEN _WarningNum := 0; END_IF

// NETWORK 2
//   Control.Outputs.Warning: Machine has a warning active
_w1 := _WarningNum <> 0;
_Warning := _w1;
_r_Trig[5](CLK := _w1); // R_TRIG
Control.Outputs.Warning S= _r_Trig[5].Q AND NOT Control.Outputs.Warning;

// NETWORK 3
//   Control.Outputs.Warning: Machine has a warning active
_r_Trig[4](CLK := _WarningNum = 0); // R_TRIG
Control.Outputs.Warning R= _r_Trig[4].Q;

// NETWORK 4
M_LogWarning(Execute := _Warning, Arg0 := _Name, Arg1 := _Description, Arg2 := '', EventEntry := M_Warnings(), Clear := NOT _Warning, Message := Control.Outputs.WarningMessage);

// NETWORK 5
IF _AlarmMute THEN _WarningNum := 2110; END_IF
END_METHOD

METHOD M_Warnings : TcEventEntry
VAR_INPUT
END_VAR
CASE _WarningNum OF
	2110: M_Warnings:= TC_Events.TcTcpIpClient.W_2110;//Alarm Mute Active				
ELSE
	M_Warnings:=  TC_Events.TcTcpIpClient.W_Undefined;	
END_CASE
END_METHOD

{attribute 'monitoring' := 'variable'}
PROPERTY PUBLIC Name : String[15]
GET
Name := _Name;
END_GET
SET
_Name := Name;
END_SET
END_PROPERTY

{attribute 'monitoring' := 'variable'}
PROPERTY PUBLIC Warning : Bool
GET
Warning := _Warning;
END_GET
END_PROPERTY

END_FUNCTION_BLOCK

// Objects/FB_TcpIpServer_V4_00/FB_TcpIpServer
FUNCTION_BLOCK FB_TcpIpServer EXTENDS FB_EventLogger 
VAR_INPUT
	Enable					: BOOL;//Enable TCP/IP Commnuication
	LocalHost				: T_IPv4Addr := '127.0.0.1';//TCP/IP Socket IP Address
	LocalPort				: UDINT := 1024;//TCP/IP Socket Port
	ReconnectTime			: TIME := T#3S;//Time until reconnection is attempted
	AcceptPollingTime		: TIME := T#100MS;//Send poll time
	RecievePollingTime		: TIME := T#100MS;//Recieve poll Time
	RecieveTimeOut			: TIME := T#3S;// Recieve timeout
	TxData					: ANY;//Raw send data
	RxData					: ANY;//Raw recieve data
	Delimiter				: BYTE := 0;//String data type delimiter in ASCII format
END_VAR                     
VAR_IN_OUT                  
	Control					: ST_System;
END_VAR                     
VAR_OUTPUT                  
	Listening				: BOOL;//Listening for inoming connections
	Accepted				: BOOL;//Socket connection accepted
	SendRecieveRate			: REAL;//Time to send and recieve data over TCP/IP.
END_VAR
VAR
	{attribute 'tc_no_symbol'}   
	_fb_Listen	 			: FB_SocketListen := ( sSrvNetID := '', tTimeout := DEFAULT_ADS_TIMEOUT );//Listener for incoming connection requests from remote clients
	{attribute 'tc_no_symbol'} 
	_fb_SocketClose			: FB_SocketClose := ( sSrvNetID := '', tTimeout := DEFAULT_ADS_TIMEOUT );//Closes an open TCP/IP or UDP socket.
	{attribute 'tc_no_symbol'} 
	_fb_RemoteSocketClose	: FB_SocketClose := ( sSrvNetID := '', tTimeout := DEFAULT_ADS_TIMEOUT );//Closes an open TCP/IP or UDP socket.
	{attribute 'tc_no_symbol'} 
	_fb_SocketAccept		: FB_SocketAccept := ( sSrvNetID := '', tTimeout := DEFAULT_ADS_TIMEOUT );//Accepts remote client connection requests
	{attribute 'tc_no_symbol'} 
	_fb_SocketSend	 		: FB_SocketSend := ( sSrvNetID := '', tTimeout := DEFAULT_ADS_TIMEOUT );//Sends data to a remote client or remote server via the TwinCAT TCP/IP
	{attribute 'tc_no_symbol'} 
	_fb_SocketReceive		: FB_SocketReceive := ( sSrvNetID := '', tTimeout := DEFAULT_ADS_TIMEOUT );//Receives data from a remote client or remote server via the TwinCAT TCP/IP
	{attribute 'tc_no_symbol'} 
	_fb_ConnectTON			: TON;					//Reconnection Timer
	_eStep					: E_ServerSteps;		//Step Engine
	_Listener 				: T_HSOCKET;			//Connection handle of an open socket
	_Alarm					: BOOL;					//Device Alarm
	_Warning				: BOOL;					//Device Warning
	_Message				: BOOL;					//Device Message
	_AlarmNum				: DINT;					//Device Alarm Number
	_WarningNum				: DINT;					//Device Warning Number
	_MessageNum				: DINT;					//Device Message Number
	_Fault					: BOOL;					//Device Fault
	_FaultTimer_ET			: REAL;					//Fault timer elapsed
	_ExtendedErrorCode		: UDINT;				//Extended Error Code
	_RecieveTimeOut			: BOOL;					//No bytes recieved in time error
	_RecieveBufferOverflow	: BOOL;					//No more free read buffer space error
	_r_Trig					: ARRAY[0..9] OF R_TRIG;//Public Rising Edge Triggers
END_VAR                 	
VAR PERSISTENT          	
	_Name					: STRING[15];			//Name for HMI
	_Description			: STRING[40];			//Description for HMI
	_AlarmMute				: BOOL;					//Alarm Mute
	_FaultTimer_PT			: REAL;					//Fault timer preset time
END_VAR

M_AlarmMonitor();
M_WarningMonitor();
M_MessageMonitor();

IF Control.Inputs.AlarmMuteReset THEN _AlarmMute := FALSE; END_IF

CASE _eStep OF

	SERVER_STATE_IDLE:
		IF Enable XOR Listening THEN
			IF Enable THEN
				_fb_ConnectTON( IN := FALSE );
				_eStep := SERVER_STATE_LISTENER_OPEN_START;
			ELSE
				SendRecieveRate := 0;
				_eStep := SERVER_STATE_REMOTE_CLIENTS_CLOSE;
			END_IF
		ELSIF Listening THEN
			_eStep := SERVER_STATE_REMOTE_CLIENTS_COMM;
		END_IF

	SERVER_STATE_LISTENER_OPEN_START:
		_fb_ConnectTON( IN := TRUE, PT := ReconnectTime );
		IF _fb_ConnectTON.Q THEN
		   _fb_ConnectTON( IN := FALSE );
		   _fb_Listen(  bExecute := FALSE  );
		   _fb_Listen(	sLocalHost	:= LocalHost, nLocalPort:= LocalPort, bExecute:= TRUE );
		    _eStep := SERVER_STATE_LISTENER_OPEN_WAIT;
		END_IF

	SERVER_STATE_LISTENER_OPEN_WAIT:
		_fb_Listen( bExecute := FALSE );
		IF NOT _fb_Listen.bBusy THEN
			IF NOT _fb_Listen.bError THEN
				Listening 	:= TRUE;
				_Listener 	:= _fb_Listen.hListener;
				_eStep 	:= SERVER_STATE_IDLE;
			ELSE
				_eStep := SERVER_STATE_ERROR;
			END_IF
		END_IF

	SERVER_STATE_REMOTE_CLIENTS_COMM:
		_eStep := SERVER_STATE_IDLE;
		IF M_RemoteClient(Enable:= TRUE, Listener := _Listener) THEN (*FB_SocketAccept returned error!*)
			_eStep := SERVER_STATE_REMOTE_CLIENTS_CLOSE;
		END_IF	
		
	SERVER_STATE_REMOTE_CLIENTS_CLOSE:
		_eStep := SERVER_STATE_LISTENER_CLOSE_START; (* close listener socket too *)
		IF NOT M_RemoteClient(Enable:= FALSE, Listener := _Listener) AND Accepted THEN
			_eStep := SERVER_STATE_REMOTE_CLIENTS_CLOSE; (* stay here and close all remote clients first *)
		END_IF
	
	SERVER_STATE_LISTENER_CLOSE_START:
		_fb_SocketClose( bExecute := FALSE );
		_fb_SocketClose(	hSocket	:= _Listener,bExecute:= TRUE );
		_eStep := SERVER_STATE_LISTENER_CLOSE_WAIT;

	SERVER_STATE_LISTENER_CLOSE_WAIT:
		_fb_SocketClose( bExecute := FALSE );
		IF NOT _fb_SocketClose.bBusy THEN
			Listening := FALSE;
			MEMSET( ADR(_Listener), 0, SIZEOF(_Listener));
			IF _fb_SocketClose.bError THEN
				_eStep := SERVER_STATE_ERROR;
			ELSE
				_eStep := SERVER_STATE_IDLE;
			END_IF
		END_IF

	SERVER_STATE_ERROR:
		IF Listening THEN
			_eStep := SERVER_STATE_REMOTE_CLIENTS_CLOSE;
		ELSE
			_eStep := SERVER_STATE_IDLE;
		END_IF

END_CASE

{attribute 'monitoring' := 'variable'}
PROPERTY PUBLIC Alarm : Bool
GET
Alarm := _Alarm;
END_GET
END_PROPERTY

{attribute 'monitoring' := 'variable'}
PROPERTY PUBLIC AlarmMute : BOOL
SET
AlarmMute := _AlarmMute;
END_SET
END_PROPERTY

{attribute 'monitoring' := 'variable'}
PROPERTY PUBLIC Description : String[40]
GET
Description := _Description;
END_GET
SET
_Description := Description;
END_SET
END_PROPERTY

{attribute 'monitoring' := 'variable'}
PROPERTY PUBLIC Fault : Bool
SET
_Fault := Fault;
END_SET
END_PROPERTY

{attribute 'monitoring' := 'variable'}
PROPERTY PUBLIC FaultTimer_PT : real
GET
FaultTimer_PT := _FaultTimer_PT;
END_GET
SET
_FaultTimer_PT := FaultTimer_PT;
END_SET
END_PROPERTY

METHOD PRIVATE M_AlarmMonitor
VAR_INPUT
END_VAR
VAR_INST
END_VAR
VAR_INST // added by the converter: edge detectors and wires of the graphical bodies
    _w1, _w2, _w3, _w4, _w5 : BOOL;
    _rt1, _rt2, _rt3, _rt4, _rt5, _rt6, _rt7, _rt8 : R_TRIG;
END_VAR
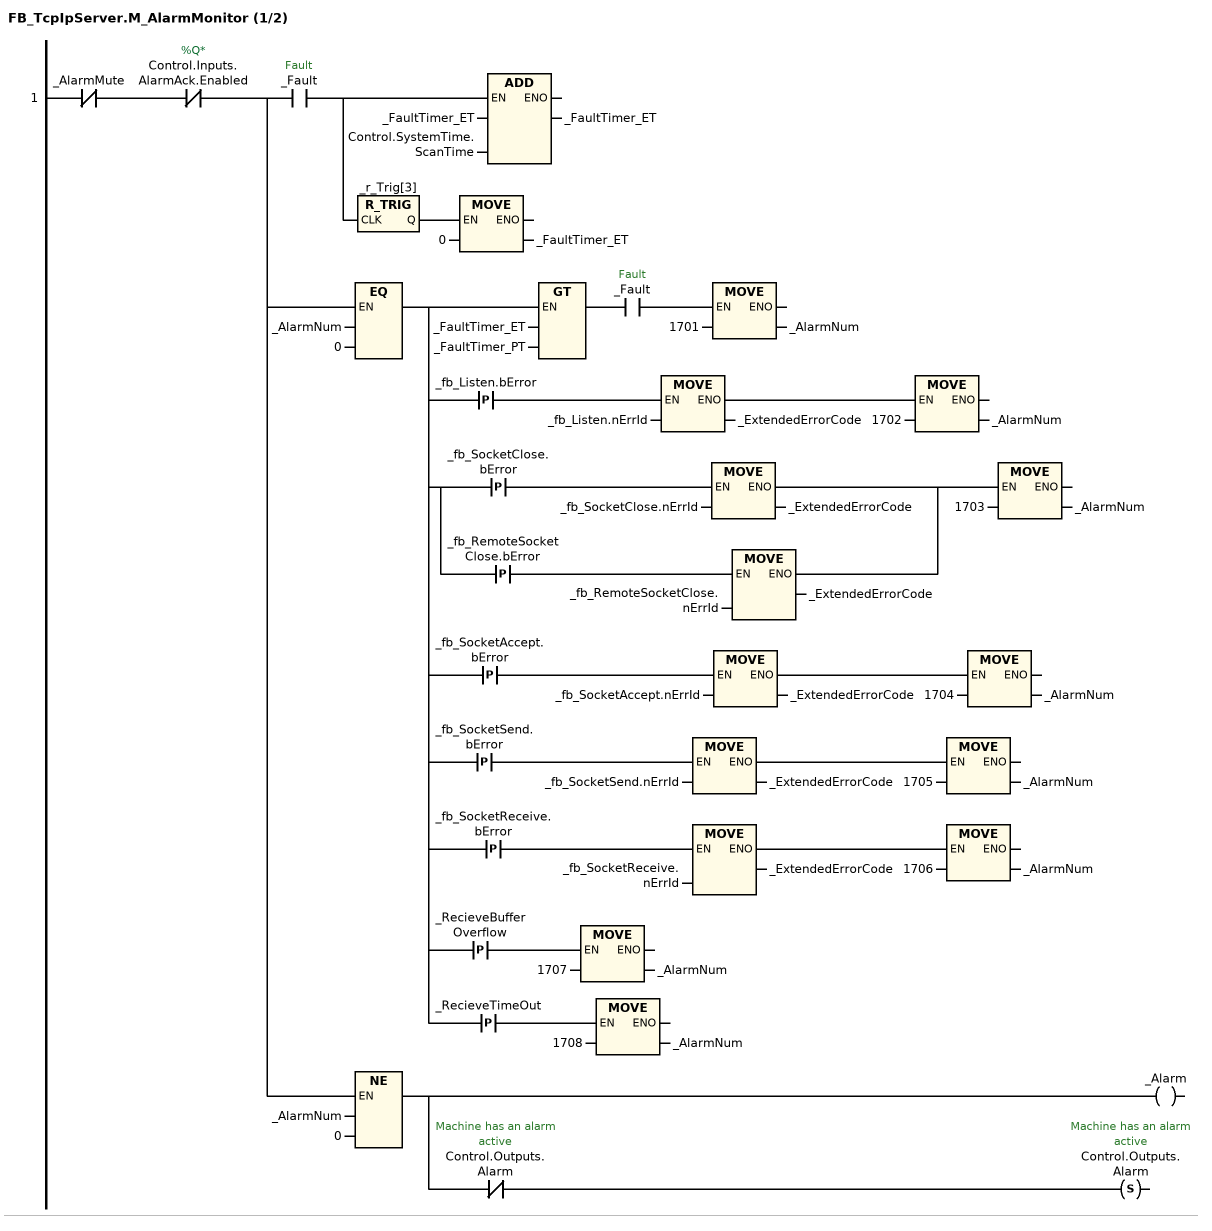
// NETWORK 1
//   Control.Inputs.AlarmAck.Enabled: AT %Q*
//   _Fault: Fault
//   _FaultTimer_ET: Fault timer elapsed
//   Control.SystemTime.ScanTime: Last scan time (Seconds)
//   _FaultTimer_PT: Fault timer preset time
//   Control.Outputs.Alarm: Machine has an alarm active
_w1 := NOT _AlarmMute AND NOT Control.Inputs.AlarmAck.Enabled;
_w2 := _w1 AND _Fault;
IF _w2 THEN _FaultTimer_ET := _FaultTimer_ET + Control.SystemTime.ScanTime; END_IF
_r_Trig[3](CLK := _w2); // R_TRIG
IF _r_Trig[3].Q THEN _FaultTimer_ET := 0; END_IF
_w3 := _w1 AND _AlarmNum = 0;
IF (_w3 AND _FaultTimer_ET > _FaultTimer_PT) AND _Fault THEN _AlarmNum := 1701; END_IF
_rt1(CLK := _fb_Listen.bError);
IF _w3 AND _rt1.Q THEN _ExtendedErrorCode := _fb_Listen.nErrId; END_IF
IF _w3 AND _rt1.Q THEN _AlarmNum := 1702; END_IF
_rt2(CLK := _fb_SocketClose.bError);
IF _w3 AND _rt2.Q THEN _ExtendedErrorCode := _fb_SocketClose.nErrId; END_IF
_rt3(CLK := _fb_RemoteSocketClose.bError);
IF _w3 AND _rt3.Q THEN _ExtendedErrorCode := _fb_RemoteSocketClose.nErrId; END_IF
IF _w3 AND _rt2.Q OR _w3 AND _rt3.Q THEN _AlarmNum := 1703; END_IF
_rt4(CLK := _fb_SocketAccept.bError);
IF _w3 AND _rt4.Q THEN _ExtendedErrorCode := _fb_SocketAccept.nErrId; END_IF
IF _w3 AND _rt4.Q THEN _AlarmNum := 1704; END_IF
_rt5(CLK := _fb_SocketSend.bError);
IF _w3 AND _rt5.Q THEN _ExtendedErrorCode := _fb_SocketSend.nErrId; END_IF
IF _w3 AND _rt5.Q THEN _AlarmNum := 1705; END_IF
_rt6(CLK := _fb_SocketReceive.bError);
IF _w3 AND _rt6.Q THEN _ExtendedErrorCode := _fb_SocketReceive.nErrId; END_IF
IF _w3 AND _rt6.Q THEN _AlarmNum := 1706; END_IF
_rt7(CLK := _RecieveBufferOverflow);
IF _w3 AND _rt7.Q THEN _AlarmNum := 1707; END_IF
_rt8(CLK := _RecieveTimeOut);
IF _w3 AND _rt8.Q THEN _AlarmNum := 1708; END_IF
_w4 := _w1 AND _AlarmNum <> 0;
_Alarm := _w4;
Control.Outputs.Alarm S= _w4 AND NOT Control.Outputs.Alarm;

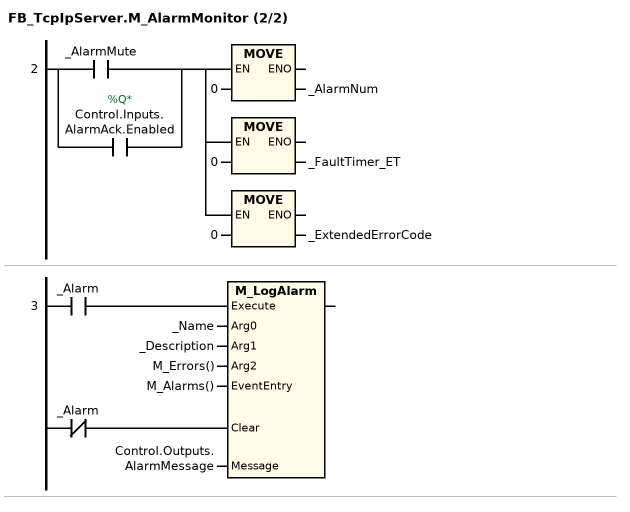
// NETWORK 2
//   Control.Inputs.AlarmAck.Enabled: AT %Q*
//   _FaultTimer_ET: Fault timer elapsed
//   _ExtendedErrorCode: Fault timer elapsed
_w5 := _AlarmMute OR Control.Inputs.AlarmAck.Enabled;
IF _w5 THEN _AlarmNum := 0; END_IF
IF _w5 THEN _FaultTimer_ET := 0; END_IF
IF _w5 THEN _ExtendedErrorCode := 0; END_IF

// NETWORK 3
M_LogAlarm(Execute := _Alarm, Arg0 := _Name, Arg1 := _Description, Arg2 := M_Errors(), EventEntry := M_Alarms(), Clear := NOT _Alarm, Message := Control.Outputs.AlarmMessage);
END_METHOD

METHOD M_Alarms : TcEventEntry
VAR_INPUT
END_VAR
CASE _AlarmNum OF
	1701: M_Alarms:= TC_Events.TcTcpIpServer.A_1701;//General error
	1702: M_Alarms:= TC_Events.TcTcpIpServer.A_1702;//Socket listen error
	1703: M_Alarms:= TC_Events.TcTcpIpServer.A_1703;//Socket close error
	1704: M_Alarms:= TC_Events.TcTcpIpServer.A_1704;//Socket accept error	
	1705: M_Alarms:= TC_Events.TcTcpIpServer.A_1705;//Socket send error	
	1706: M_Alarms:= TC_Events.TcTcpIpServer.A_1706;//Socket recieve error	
	1707: M_Alarms:= TC_Events.TcTcpIpServer.A_1707;//Receive buffer overflow
	1708: M_Alarms:= TC_Events.TcTcpIpServer.A_1708;//Receive timeout error
ELSE
	M_Alarms:= TC_Events.TcTcpIpServer.A_Undefined;
END_CASE
END_METHOD

METHOD PRIVATE M_DataExchange : BOOL;
VAR_INPUT
	Socket				: T_HSOCKET;
	Execute				: BOOL;
END_VAR             	
VAR_INST
	{attribute 'tc_no_symbol'} 
	_Busy				: BOOL;
	{attribute 'tc_no_symbol'} 
	_Error 				: BOOL;
	{attribute 'tc_no_symbol'} 
	_eStep				: E_ServerDataExchangeSteps;
	{attribute 'tc_no_symbol'} 
	_fb_ReceiveTON		: TON;
	{attribute 'tc_no_symbol'} 
	_fb_DisconnectTON 	: TON;
	{attribute 'tc_no_symbol'} 
	_cbFrame			: UDINT;
	{attribute 'tc_no_symbol'} 
	_rxBuffer			: ARRAY[0..255] OF BYTE;
	{attribute 'tc_no_symbol'} 
	_SendRecieveRate	: REAL;
	{attribute 'tc_no_symbol'} 
	_cbReceived, _startPos, _endPos, _idx	: UDINT;
END_VAR
_r_Trig[9]( CLK := Execute );
IF _SendRecieveRate > SendRecieveRate THEN SendRecieveRate :=  _SendRecieveRate; END_IF
_SendRecieveRate := _SendRecieveRate + Control.SystemTime.ScanTime;
CASE _eStep OF

	SERVER_DATAEXCHANGE_STATE_IDLE:
		IF _r_Trig[9].Q THEN
			_SendRecieveRate := 0;
			_Busy 	:= TRUE;
			_Error 	:= FALSE;
			_fb_DisconnectTON( IN := FALSE, PT := T#0MS );(* disable timeout check first *)
			_fb_ReceiveTON( IN := FALSE, PT := T#0MS ); (* receive first request immediately *)
			_eStep 	:= SERVER_DATAEXCHANGE_STATE_RECEIVE_START;
		END_IF

	SERVER_DATAEXCHANGE_STATE_RECEIVE_START: (* Receive remote client data *)
		_fb_ReceiveTON(  IN := TRUE );
		IF _fb_ReceiveTON.Q THEN
			_fb_ReceiveTON( IN := FALSE );
			_fb_SocketReceive( bExecute := FALSE );
			MEMSET(ADR( _rxBuffer ),0,SIZEOF( _rxBuffer ));
			IF RxData.TypeClass = DINT_TO_UDINT(IBaseLibrary.TYPE_STRING) THEN
				_fb_SocketReceive( hSocket:= Socket,pDest:= ADR( _rxBuffer ) , cbLen	:= SIZEOF( _rxBuffer ),bExecute	:= TRUE );
			ELSE
				_fb_SocketReceive( hSocket:= Socket,pDest := RxData.pValue, cbLen:=DINT_TO_UDINT(RxData.diSize),bExecute	:= TRUE );
			END_IF
			_eStep := SERVER_DATAEXCHANGE_STATE_RECEIVE_WAIT;
		END_IF

	SERVER_DATAEXCHANGE_STATE_RECEIVE_WAIT:
		_fb_SocketReceive( bExecute := FALSE );
		IF NOT _fb_SocketReceive.bBusy THEN
			IF NOT _fb_SocketReceive.bError THEN

				IF (_fb_SocketReceive.nRecBytes > 0) THEN(* bytes received *)

					IF RxData.TypeClass = DINT_TO_UDINT(IBaseLibrary.TYPE_STRING) THEN
						_startPos 	:= _cbReceived;(* rxBuffer array index of first data byte *)
						_endPos  	:= _cbReceived + _fb_SocketReceive.nRecBytes  - 1;(* rxBuffer array index of last data byte *)
						_cbReceived 	:= _cbReceived + _fb_SocketReceive.nRecBytes;(* calculate the number of received data bytes *)
						_cbFrame	:= 0;(* reset frame length *)
                	
						IF _cbReceived < DINT_TO_UDINT(RxData.diSize) THEN (* no overflow *)
                	
							_fb_ReceiveTON( IN := FALSE, PT := T#0S ); (* bytes received => increase the read (polling) speed *)
							_fb_DisconnectTON( IN := FALSE, PT := RecieveTimeOut);(* bytes received => disable timeout check *)
                	
							(* search for string end delimiter *)
							FOR _idx := _startPos TO _endPos BY 1 DO
								IF _rxBuffer[_idx] = Delimiter THEN(* string end delimiter found *)
									_cbFrame := _idx + 1;(* calculate the length of the received string (inclusive the end delimiter) *)
									MEMCPY(  RxData.pValue, ADR( _rxBuffer ), _cbFrame );(* copy the received string to the output variable (inclusive the end delimiter) *)
									MEMMOVE( ADR( _rxBuffer ), ADR( _rxBuffer[_cbFrame] ),  _cbReceived - _cbFrame  );(* move the reamaining data bytes *)
									_cbReceived := _cbReceived - _cbFrame;(* recalculate the reamaining data byte length *)
									_eStep := SERVER_DATAEXCHANGE_STATE_SEND_START;
									EXIT;
								END_IF
							END_FOR
                	
						ELSE(* there is no more free read buffer space => the answer string should be terminated *)
							_RecieveBufferOverflow := TRUE;
							_eStep := SERVER_DATAEXCHANGE_STATE_ERROR;
						END_IF
					ELSE
						_eStep := SERVER_DATAEXCHANGE_STATE_SEND_START;
					END_IF

				ELSE(* no bytes received *)
					_fb_ReceiveTON( IN := FALSE, PT := RecievePollingTime);(* no bytes received => decrease the read (polling) speed *)
					_fb_DisconnectTON( IN := TRUE, PT := RecieveTimeOut );(* no bytes received => enable timeout check*)
					IF _fb_DisconnectTON.Q THEN (* timeout error*)
						_fb_DisconnectTON( IN := FALSE );
						_RecieveTimeOut:= TRUE;
						_eStep := SERVER_DATAEXCHANGE_STATE_ERROR;
					ELSE(* repeat reading *)
						_eStep := SERVER_DATAEXCHANGE_STATE_RECEIVE_START; (* repeat reading *)
					END_IF
				END_IF
			ELSE(* receive error *)
				_eStep := SERVER_DATAEXCHANGE_STATE_ERROR;
			END_IF
		END_IF

	SERVER_DATAEXCHANGE_STATE_SEND_START:
		_fb_SocketSend( bExecute := FALSE );
		_fb_SocketSend(	hSocket	:= Socket,pSrc	:= TxData.pValue,cbLen	:=DINT_TO_UDINT(TxData.diSize),bExecute:= TRUE );
		_eStep := SERVER_DATAEXCHANGE_STATE_SEND_WAIT;

	SERVER_DATAEXCHANGE_STATE_SEND_WAIT:
		_fb_SocketSend( bExecute := FALSE );
		IF NOT _fb_SocketSend.bBusy THEN
			IF NOT _fb_SocketSend.bError THEN
				_Busy := FALSE;
				_eStep := SERVER_DATAEXCHANGE_STATE_IDLE;
			ELSE
				_eStep := SERVER_DATAEXCHANGE_STATE_ERROR;
			END_IF
		END_IF

	SERVER_DATAEXCHANGE_STATE_ERROR:
		_Busy := FALSE;
		_RecieveTimeOut:= FALSE;
		_RecieveBufferOverflow := FALSE;
		_Error := TRUE;
		_SendRecieveRate := 0;
		_cbReceived := 0;
		_eStep := SERVER_DATAEXCHANGE_STATE_IDLE;
END_CASE

M_DataExchange:= _Busy;
END_METHOD

METHOD PRIVATE M_Errors : STRING(126)
VAR_INPUT
END_VAR
VAR_INST
END_VAR
CASE _ExtendedErrorCode OF	
//Global Error Codes
0	: M_Errors :='';
1	: M_Errors :='1 Internal error';	 	 
2	: M_Errors :='2 No Rtime';	 	 
3	: M_Errors :='3	Allocation locked memory error';	 	 
4	: M_Errors :='4	Insert mailbox error';
5	: M_Errors :='5	Wrong receive HMSG';	 	 
6	: M_Errors :='6	target port not found	ADS Server not started';	 
7	: M_Errors :='7	target machine not found Missing ADS routes';	 
8	: M_Errors :='8	Unknown command ID';	 	 
9	: M_Errors :='9	Bad task ID';	 	 
10	: M_Errors :='10 No IO';	 	 
11	: M_Errors :='11 Unknown ADS command';	 	 
12	: M_Errors :='12 Win 32 error';	 	 
13	: M_Errors :='13 Port not connected';	 	 
14	: M_Errors :='14 Invalid ADS length';	 	 
15	: M_Errors :='15 Invalid AMS Net ID';	 	 
16	: M_Errors :='16 Low Installation level';	 	 
17	: M_Errors :='17 No debug available';	 	 
18	: M_Errors :='18 Port disabled';	 	 
19	: M_Errors :='19 Port already connected';	 	 
20	: M_Errors :='20 ADS Sync Win32 error';	 	 
21	: M_Errors :='21 ADS Sync Timeout';	 	 
22	: M_Errors :='22 ADS Sync AMS error';	 	 
23	: M_Errors :='23 ADS Sync no index map';	 	 
24	: M_Errors :='24 Invalid ADS port';	 	 
25	: M_Errors :='25 No memory';	 	 
26	: M_Errors :='26 TCP send error';	 	 
27	: M_Errors :='27 Host unreachable'; 	 
28	: M_Errors :='28 Invalid AMS fragment';
//Router Error Codes
1280 :	M_Errors :='1280 No locked memory can be allocated'; 
1281 :	M_Errors :='1281 The size of the router memory could not be changed'; 	 
1282 :	M_Errors :='1282 The mailbox has reached the maximum number OF possible messages'; 
1283 :	M_Errors :='1283 The mailbox has reached the maximum number OF possible messages'; 
1284 :	M_Errors :='1284 The port type is unknown'; 	 
1285 :	M_Errors :='1285 Router is not initialised'; 	 
1286 :	M_Errors :='1286 The desired port number is already assigned'; 	 
1287 :	M_Errors :='1287 Port not registered'; 	 
1288 :	M_Errors :='1288 The maximum number of Ports reached'; 	 
1289 :	M_Errors :='1289 The port is invalid'; 	 
1290 :	M_Errors :='1290 TwinCAT Router not active';  
1291 :	M_Errors :='1291 ROUTERERR_FRAGMENTBOXFULL'; 	 	 
1292 :	M_Errors :='1292 ROUTERERR_FRAGMENTTIMEOUT'; 	 	 
1293 :	M_Errors :='1293 ROUTERERR_TOBEREMOVED'; 
//General ADS Error Codes
1792: M_Errors :='1792 error class <device error>';	 	 
1793: M_Errors :='1793 Service is not supported by server';	 	 
1794: M_Errors :='1794 invalid index group';	 	 
1795: M_Errors :='1795 invalid index offset';	 	 
1796: M_Errors :='1796 reading/writing not permitted';	 	 
1797: M_Errors :='1797 parameter size not correct';	 	 
1798: M_Errors :='1798 invalid parameter value(S)';	 	 
1799: M_Errors :='1799 device is not in a ready state';	 	 
1800: M_Errors :='1800 device is busy';	 	 
1801: M_Errors :='1801 invalid context (must be in Windows)';	 	 
1802: M_Errors :='1802 out OF memory';	 	 
1803: M_Errors :='1803 invalid parameter value(s)';	 	 
1804: M_Errors :='1804 not found (files, ...)';	 	 
1805: M_Errors :='1805 syntax error in command or file';	 	 
1806: M_Errors :='1806 objects DO not match';	 	 
1807: M_Errors :='1807 object already exists';	 	 
1808: M_Errors :='1808 symbol not found';	 	 
1809: M_Errors :='1809 symbol version invalid';	
1810: M_Errors :='1810 server is in invalid state';	 	 
1811: M_Errors :='1811 AdsTransMode not supported';	 	 
1812: M_Errors :='1812 notification handle is invalid';	
1813: M_Errors :='1813 notification client not registered';	 	 
1814: M_Errors :='1814 no more notification handles';	 	 
1815: M_Errors :='1815 size for watch too big';	 	 
1816: M_Errors :='1816 device not initialized';	 	 
1817: M_Errors :='1817 device has a timeout';	 	 
1818: M_Errors :='1818 query INTERFACE failed';	 	 
1819: M_Errors :='1819 wrong interface required';	 	 
1820: M_Errors :='1820 class ID is invalid';	 	 
1821: M_Errors :='1821 object ID is invalid';	 	 
1822: M_Errors :='1822 request is pending';	 	 
1823: M_Errors :='1823 request is aborted';	 	 
1824: M_Errors :='1824 signal warning';	 	 
1825: M_Errors :='1825 invalid array index';	 	 
1826: M_Errors :='1826 symbol not active';	
1827: M_Errors :='1827 access denied';	 	 
1828: M_Errors :='1828 missing license';	 	
1836: M_Errors :='1836 exception occured during system start';	
1856: M_Errors :='1856 Error class <client error>';	 	 
1857: M_Errors :='1857 invalid parameter at service';	 	 
1858: M_Errors :='1858 polling list is empty';	 	 
1859: M_Errors :='1859 var connection already in use';	 	 
1860: M_Errors :='1860 invoke ID in use';	 	 
1861: M_Errors :='1861 timeout elapsed'; 	
1862: M_Errors :='1862 error in win32 subsystem';	 	 
1863: M_Errors :='1863 Invalid client timeout value';	 	 
1864: M_Errors :='1864 ads-port not opened';	 	 
1872: M_Errors :='1872 internal error in ads sync';	 	 
1873: M_Errors :='1873 hash table overflow';	 	 
1874: M_Errors :='1874 key not found in hash';	 	 
1875: M_Errors :='1875 no more symbols in cache';	 	 
1876: M_Errors :='1876 invalid response received';	 	 
1877: M_Errors :='1877 sync port is locked';
//RTime Error Codes
4096: M_Errors:= '4096 INTERNAL error in the REAL-TIME system.';
4097: M_Errors:= '4097 Timer value is NOT valid.';
4098: M_Errors:= '4098 Task pointer has the invalid value 0 (zero).';
4099: M_Errors:= '4099 Stack POINTER has the invalid value 0 (zero).';
4100: M_Errors:= '4100 The request task priority is already assigned.';
4101: M_Errors:= '4101 No free TCB (Task Control Block) available. The maximum number OF TCBs is 64.';
4102: M_Errors:= '4102 No free semaphores available. The maximum number of semaphores is 64.';
4103: M_Errors:= '4103 No free space available in the queue. The maximum number OF positions in the queue is 64.';
4109: M_Errors:= '4109 An external synchronization interrupt is already applied.';
4110: M_Errors:= '4110 No external sync interrupt applied.';
4111: M_Errors:= '4111 Application of the external synchronization interrupt has failed.';
4112: M_Errors:= '4112 Call OF a service FUNCTION in the wrong context';
4119: M_Errors:= '4119 Intel VT-x extension is not supported.';
4120: M_Errors:= '4120 Intel VT-x extension is NOT enabled in the BIOS.';
4121: M_Errors:= '4121 Missing function in Intel VT-x extension.';
4122: M_Errors:= '4122 Activation OF Intel VT-x fails.';
//TCP Winsock Error Codes
10060: M_Errors:= '10060 Intel VT-x extension is NOT enabled in the BIOS.';
10061: M_Errors:= '10061 Missing function in Intel VT-x extension.';
10065: M_Errors:= '10065 Activation OF Intel VT-x fails.';
//Internal error codes of the TwinCAT TCP/IP Connection Server
32769: M_Errors:= '32769 No new sockets can be created (for FB_SocketListen AND FB_SocketConnect).';
32770: M_Errors:= '32770 Socket handle is invalid (for FB_SocketReceive, FB_SocketAccept, FB_SocketSend etc.).';
32771: M_Errors:= '32771 Is returned when FB_SocketListen is called, if the TcpIp port listener already exists.';
32772: M_Errors:= '32772 Is returned when FB_SocketReceive is called, if the client socket is no longer connected with the server.';
32773: M_Errors:= '32773 Is returned when FB_SocketAccept is called, if an error was registered in the listener socket.';
//Internal SNMP error codes
36865: M_Errors:= '36865 INCORRECT PARAMETER SIZE';
36866: M_Errors:= '36866 INVALID PARAMETER';
ELSE
	M_Errors := 	CONCAT('Undefined TCP Server Error - ' , TO_STRING( _ExtendedErrorCode));
END_CASE
END_METHOD

METHOD PRIVATE M_MessageMonitor
VAR_INPUT
END_VAR
VAR_INST
END_VAR
VAR_INST // added by the converter: edge detectors and wires of the graphical bodies
    _w1 : BOOL;
    _rt1, _rt2 : R_TRIG;
    _ft1, _ft2 : F_TRIG;
END_VAR
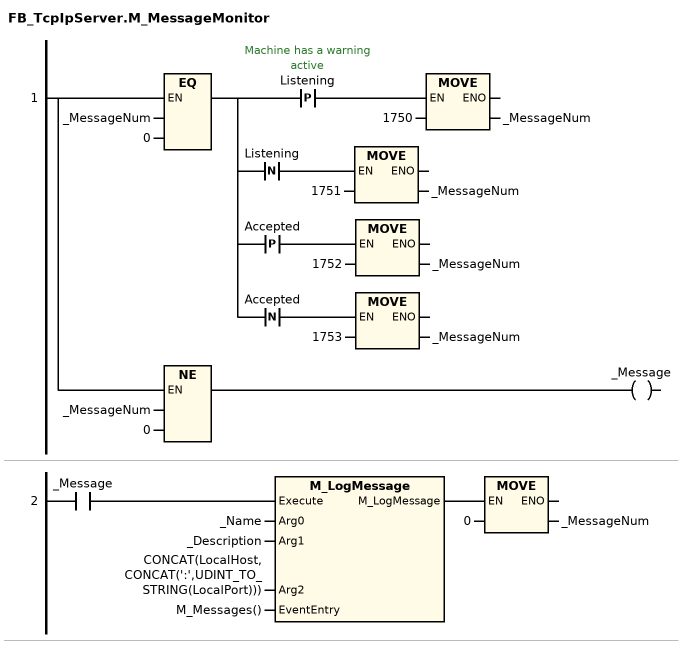
// NETWORK 1
//   Listening: Machine has a warning active
_w1 := _MessageNum = 0;
_rt1(CLK := Listening);
IF _w1 AND _rt1.Q THEN _MessageNum := 1750; END_IF
_ft1(CLK := Listening);
IF _w1 AND _ft1.Q THEN _MessageNum := 1751; END_IF
_rt2(CLK := Accepted);
IF _w1 AND _rt2.Q THEN _MessageNum := 1752; END_IF
_ft2(CLK := Accepted);
IF _w1 AND _ft2.Q THEN _MessageNum := 1753; END_IF
_Message := _MessageNum <> 0;

// NETWORK 2
IF M_LogMessage(Execute := _Message, Arg0 := _Name, Arg1 := _Description, Arg2 := CONCAT(LocalHost,CONCAT(':',UDINT_TO_STRING(LocalPort))), EventEntry := M_Messages()) THEN
    _MessageNum := 0;
END_IF
END_METHOD

METHOD PRIVATE M_Messages : TcEventEntry
VAR_INPUT
END_VAR
CASE _MessageNum OF
	1750: M_Messages:= TC_Events.TcTcpIpServer.M_1750;//Listener socket open
	1751: M_Messages:= TC_Events.TcTcpIpServer.M_1751;//Listener socket closed
	1752: M_Messages:= TC_Events.TcTcpIpServer.M_1752;//Remote client accepted
	1753: M_Messages:= TC_Events.TcTcpIpServer.M_1753;//Remote client closed	
END_CASE
END_METHOD

METHOD PRIVATE M_RemoteClient : BOOL;
VAR_INPUT
	Enable 				: BOOL;
	Listener			: T_HSOCKET;
END_VAR
VAR_INST
	{attribute 'tc_no_symbol'} 
	_Busy				: BOOL;
	{attribute 'tc_no_symbol'} 
	_Error 				: BOOL;
	{attribute 'tc_no_symbol'} 
	_HSocket			: T_HSOCKET;
	{attribute 'tc_no_symbol'} 
	_fb_SocketAcceptTON	: TON;
	{attribute 'tc_no_symbol'} 
	_eStep				: E_ClientSteps;		
END_VAR
CASE _eStep OF

	CLIENT_STATE_IDLE:
		IF Enable XOR Accepted THEN
			_Busy := TRUE;
			_Error := FALSE;
			IF Enable THEN
				_fb_SocketAcceptTON( IN := FALSE );
				_eStep := CLIENT_STATE_CONNECT_START;
			ELSE
				_eStep := CLIENT_STATE_CLOSE_START;
			END_IF
		ELSIF Accepted THEN
			_eStep := CLIENT_STATE_DATAEXCHANGE_START;
		ELSE
			_Busy := FALSE;
		END_IF

	CLIENT_STATE_CONNECT_START:
		_fb_SocketAcceptTON( IN := TRUE, PT := AcceptPollingTime);
		IF _fb_SocketAcceptTON.Q THEN
			_fb_SocketAcceptTON( IN := FALSE );
			_fb_SocketAccept(bExecute := FALSE  );
			_fb_SocketAccept(hListener := Listener,bExecute:= TRUE );
			_eStep := CLIENT_STATE_CONNECT_WAIT;
		END_IF

	CLIENT_STATE_CONNECT_WAIT:
		_fb_SocketAccept( bExecute := FALSE );
		IF NOT _fb_SocketAccept.bBusy THEN
			IF NOT _fb_SocketAccept.bError THEN
				IF _fb_SocketAccept.bAccepted THEN
					Accepted := TRUE;
					_HSocket := _fb_SocketAccept.hSocket;
				END_IF
				_eStep := CLIENT_STATE_IDLE;
			ELSE
				_eStep := CLIENT_STATE_ERROR;
			END_IF
		END_IF

	CLIENT_STATE_DATAEXCHANGE_START:
		M_DataExchange( Execute := FALSE,Socket := _HSocket);
		M_DataExchange( Execute := TRUE ,Socket :=_HSocket);
		_eStep := CLIENT_STATE_DATAEXCHANGE_WAIT;

	CLIENT_STATE_DATAEXCHANGE_WAIT:	
		IF NOT M_DataExchange( Execute := FALSE,Socket := _HSocket) THEN
			_eStep := CLIENT_STATE_IDLE;
		END_IF

	CLIENT_STATE_CLOSE_START:
		_fb_RemoteSocketClose( bExecute := FALSE );
		_fb_RemoteSocketClose(hSocket:= _HSocket,bExecute:= TRUE );
		_eStep := CLIENT_STATE_CLOSE_WAIT;

	CLIENT_STATE_CLOSE_WAIT:
		_fb_RemoteSocketClose( bExecute := FALSE );
		IF NOT _fb_RemoteSocketClose.bBusy THEN
			Accepted := FALSE;
			MEMSET( ADR( _HSocket ),0, SIZEOF( _HSocket ));
			IF _fb_RemoteSocketClose.bError THEN
				_eStep := CLIENT_STATE_ERROR;
			ELSE
				_Busy := FALSE;
				_Error := FALSE;
				_eStep := CLIENT_STATE_IDLE;
			END_IF	
		END_IF

	CLIENT_STATE_ERROR:
		_Error := TRUE;
		IF Accepted THEN
			_eStep := CLIENT_STATE_CLOSE_START;
		ELSE
			_eStep := CLIENT_STATE_IDLE;
			_Busy := FALSE;
		END_IF

END_CASE

M_RemoteClient:= NOT _Busy AND _Error;
END_METHOD

METHOD PRIVATE M_WarningMonitor
VAR_INPUT
END_VAR
VAR_INST
END_VAR
VAR_INST // added by the converter: edge detectors and wires of the graphical bodies
    _w1 : BOOL;
END_VAR
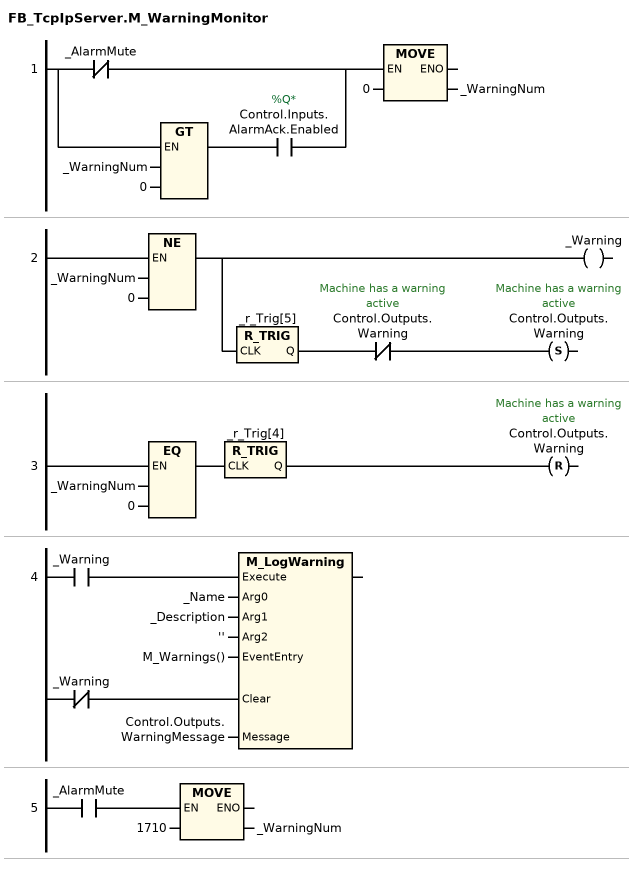
// NETWORK 1
//   Control.Inputs.AlarmAck.Enabled: AT %Q*
IF NOT _AlarmMute OR _WarningNum > 0 AND Control.Inputs.AlarmAck.Enabled THEN _WarningNum := 0; END_IF

// NETWORK 2
//   Control.Outputs.Warning: Machine has a warning active
_w1 := _WarningNum <> 0;
_Warning := _w1;
_r_Trig[5](CLK := _w1); // R_TRIG
Control.Outputs.Warning S= _r_Trig[5].Q AND NOT Control.Outputs.Warning;

// NETWORK 3
//   Control.Outputs.Warning: Machine has a warning active
_r_Trig[4](CLK := _WarningNum = 0); // R_TRIG
Control.Outputs.Warning R= _r_Trig[4].Q;

// NETWORK 4
M_LogWarning(Execute := _Warning, Arg0 := _Name, Arg1 := _Description, Arg2 := '', EventEntry := M_Warnings(), Clear := NOT _Warning, Message := Control.Outputs.WarningMessage);

// NETWORK 5
IF _AlarmMute THEN _WarningNum := 1710; END_IF
END_METHOD

METHOD M_Warnings : TcEventEntry
VAR_INPUT
END_VAR
CASE _WarningNum OF
	1710: M_Warnings:= TC_Events.TcTcpIpServer.W_1710;//Alarm Mute Active				
ELSE
	M_Warnings:=  TC_Events.TcTcpIpServer.W_Undefined;	
END_CASE
END_METHOD

{attribute 'monitoring' := 'variable'}
PROPERTY PUBLIC Name : String[15]
GET
Name := _Name;
END_GET
SET
_Name := Name;
END_SET
END_PROPERTY

{attribute 'monitoring' := 'variable'}
PROPERTY PUBLIC Warning : Bool
GET
Warning := _Warning;
END_GET
END_PROPERTY

END_FUNCTION_BLOCK

// Objects/FB_TimeManagement_V4_00/FB_TimeManagement
FUNCTION_BLOCK FINAL FB_TimeManagement
VAR_IN_OUT
	Control				: ST_System;
	Control_SP			: ST_System_SP;
END_VAR
VAR
	_fb_CurrentTicks	: GETCPUCOUNTER;
	_fb_LocalSystemTime	: FB_LocalSystemTime;
	_CurrentScan		: DWORD := 0;
	_LastScan			: DWORD := 0;
	_LastScanTime		: DWORD := 0;
	_Timer_ET			: DINT;
	_Firstscan			: R_TRIG;
	_MinutePulse		: R_TRIG;
	_HourPulse			: R_TRIG;
	_fb_GetThisTaskIdx	: GETCURTASKINDEX;
	_TaskIndex			: BYTE;
	_TaskCycleCount		: UDINT;
	_TaskCycleCountLast	: UDINT;
	_TaskStarting		: BOOL;
	_StrobeTimer		: TON;
END_VAR
VAR CONSTANT
	_ticksInSecond		: DINT := 10000000;
END_VAR

A_FirstCycle();
A_LastScanTime();
A_Strobes();
A_SyncSystemTime();
A_TimePulses();
A_UpTime();

ACTION A_FirstCycle:
_fb_GetThisTaskIdx(INDEX => _TaskIndex);
_TaskCycleCount := _TaskInfo[BYTE_TO_INT(_TaskIndex)].CycleCount;

IF _TaskCycleCount > (_TaskCycleCountLast+100) THEN
	_TaskStarting := 1;
ELSE
	_TaskStarting := 0;	
END_IF
_TaskCycleCountLast := _TaskCycleCount;

_firstscan(CLK:=_TaskStarting);

IF _firstscan.Q THEN
	Control.SystemTime.FirstCycle := TRUE;
ELSE
	Control.SystemTime.FirstCycle := FALSE;
END_IF
END_ACTION

ACTION A_LastScanTime:
_fb_CurrentTicks();
_currentScan := _fb_CurrentTicks.cpuCntLoDW;

IF _lastScan > 0 THEN
	_lastScanTime := _currentScan - _lastScan;
	//Convert to seconds
	Control.SystemTime.ScanTime := DWORD_TO_REAL(_lastScanTime) / DINT_TO_REAL(_ticksInSecond);
END_IF

_lastScan := _currentScan;
END_ACTION

ACTION A_Strobes:
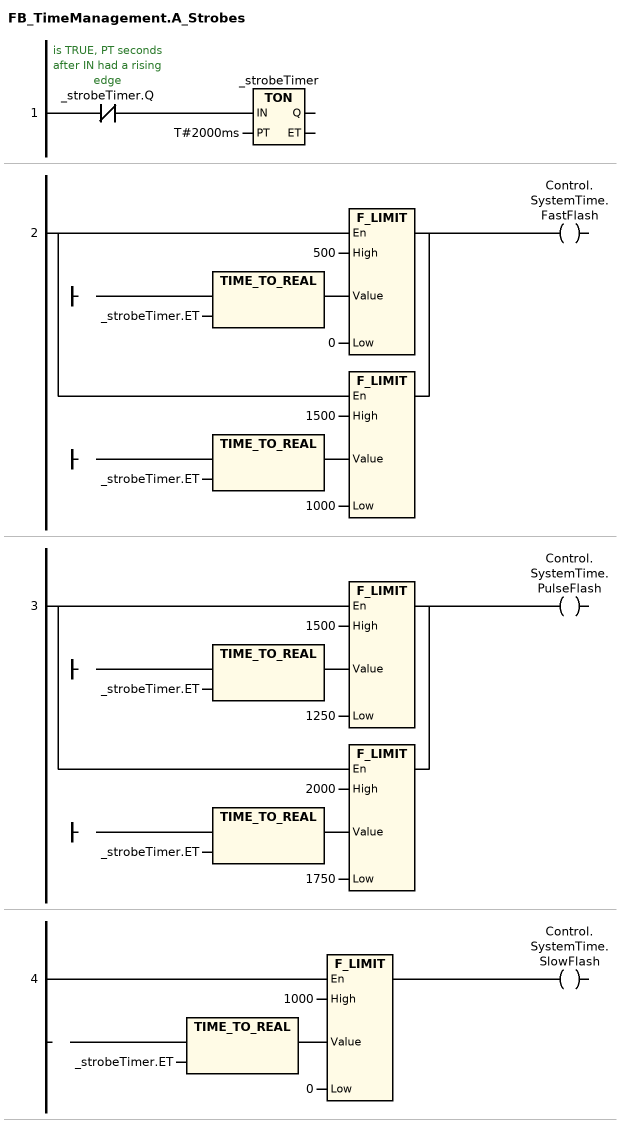
// NETWORK 1
//   _strobeTimer.Q: is TRUE, PT seconds after IN had a rising edge
_strobeTimer(IN := NOT _strobeTimer.Q, PT := T#2000ms); // TON

